IF rtbTrigger.Q OR bKeepTryingMove OR bTriggerCounter THEN
		bTriggerCounter := FALSE; 
		bKeepTryingMove := FALSE;
		nFormCounter := 0;
		bBottlePresent:= bCapPresent  := FALSE; 
		
			FOR j:=1 TO 3 DO
				FOR i:= 1 TO iExitArrayElements-1 DO // SORTOWANIE
					IF NOT eExitState[i].bFormPresent THEN 
						eExitState[i] := eExitState[i+1];
						eExitState[i+1] := eClearPackageState;
					END_IF
				END_FOR
			END_FOR	
		
			FOR i := 1 TO iEntranceArrayElements DO
				IF  NOT eExitState[i].bFormPresent THEN  		// Jeżeli w rejestrze wyjściowym jest wolne miejsce to wpisz rejestr wejściowy
					eExitState[i] := eEntranceState[1];	// Wpisz do rejestru dane np z [1] Buffor do [1,2,3,4,5,6] Package
					eEntranceState[1]:=eClearPackageState;	// Czyszczenie pierwszego rejestru wejściowego
					k:=i;											// Przepisywanie zmiennej pomocniczej
					FOR i := 1 TO iEntranceArrayElements DO   				
						IF i = iEntranceArrayElements THEN
							eEntranceState[i]:=eClearPackageState;		  // Zerowanie ostatniego bo zostało przesuniete wszystko o 1
						ELSE													  // Przepisanie 2 do 1, 3 do 2, 4 do 3, 5 do 4, 6 do 5, zeruj 6
							eEntranceState[i] := eEntranceState[i+1]; // 2 do 1, 3 do 2,
							eEntranceState[i+1]:=eClearPackageState;		  // zeruj 2, 
						END_IF
					END_FOR
					bTriggerDone := TRUE;
					EXIT;
					bError := TRUE;
					iError := 1;
				ELSE
					nFormCounter := nFormCounter + 1;
					bError := TRUE;
					iError := 2;
				END_IF
			END_FOR
		
		IF nFormCounter = iExitArrayElements THEN
		bKeepTryingMove:=NOT bNoKeepTryingMove;
		END_IF
	END_IF


//CZYSZCZENIE REJESTRU WEJSCIOWEGO
IF rtbReset.Q THEN
	FOR r1 := 1 TO iEntranceArrayElements DO
		eEntranceState[r1] := eClearPackageState;
	END_FOR
	FOR r2 := 1 TO iExitArrayElements DO
		eExitState[r2] := eClearPackageState;
	END_FOR
	bKeepTryingMove :=FALSE;
	bTriggerDone := FALSE;
	bTriggerCounter := FALSE; 
	nFormCounter := 0;
	bBottlePresent := bCapPresent := FALSE; 
	bError := FALSE;
	iError := 0;
END_IF

END_FUNCTION_BLOCK

// ---- POUs/FB/FB_InputFilter_v2.TcPOU
(*
Nazwa:			FB_InputFilter_v2
Opis: 			Filtrowanie czujnikow
Wersja:			v1.1
Data:			2023-09-20
Autor:			DP
Urzadzenia:		
Konfiguracja:	
Info:
- blok filtrujacy wejście cyfrowe
*)

FUNCTION_BLOCK FB_InputFilter_v2
VAR_INPUT
	bIN:BOOL;				//Wejście cyfrowe
	tFilterTimeOn:TIME;		//Czas filtrowania
	tFilterTimeOff:TIME;	//Czas filtrowania
END_VAR
VAR_OUTPUT
	bOUT:BOOL;
END_VAR
VAR
	tonIN: TON;
	tonOFF: TON;
END_VAR


(* w2 *)
tonIN	(IN:=bIN, 		PT:=tFilterTimeOn);
tonOFF	(IN:=NOT bIN, 	PT:=tFilterTimeOff);
IF tonIN.Q THEN
	bOUT := 	TRUE;
ELSIF tonOFF.Q THEN
	bOUT := 	FALSE;
END_IF

END_FUNCTION_BLOCK

// ---- POUs/FB/FB_MoveRegisterSortAndMoveROPP.TcPOU
(*
Nazwa:			FB_MoveRegister
Opis:			Blok przesuniecia rejestru formatek
Wersja:			v0.3 		
Data:			2018-11-16
Autor:			DP
Urzadzenia:		 
Konfiguracja:	
Info:
- Są dwa rejestry, wejściowy i wyjsciowy (struktury)
- Jezeli rejestr ma np. 6 elementów to za kazdym razem po wykryciu trigera program będzie
	1 wejściowy przesuwał na 1 wolny (nie ma formatki) wyjściowy
	kasował 1 rejestr wejściowy
	przesuwal rejetr wejsciowy 2 na 1(przeniesiony i skasowany), 3 na 2, 4 na 3, 5 na 4, 6 na 5 i kasowal 6wejsciowy
	tym sposobem po 6 trigerach caly rejestr wejsciowy powinien być na wyjsciowym
	np po 3 trigerach na wyjsciowym powinny byc zajete 1 do 3 i na wejsciowym 1 do 3
Błędy:
1 - nie wyszło z pętli for
2 - formatka już jest w rejestrze
Uwagi:
- 
Zmiany:
2018-09-18 Dodano sprawdzanie nasadek
2018-06-14 DP Pierwsza wersja
*)

FUNCTION_BLOCK FB_MoveRegisterSortAndMoveROPP
VAR_INPUT
	bFirstCycle:BOOL;					//Pierwszy cykl, zeby na początku nie wykrywało zbocza opadającego
	bTrigger :BOOL;						// Przesuniecie tablicy o jeden
	tTriggerFilterTimeOn:TIME:=T#0MS;	// Czas filtrowania wejścia Trigger na załączenie
	tTriggerFilterTimeOff:TIME:=T#0MS;	// Czas filtrowania wejścia Trigger na wyłączenie
	bTriggerBottle :BOOL;				// Zapisywanie czy jest butelka czy nie (jezeli kontrola wlączona)
	bWithBottleControl: BOOL;			// Włączona opcja kontroli butelek
	bWithCapControl:BOOL;				// Wlaczona kontrola nasadek
	bWithFormControlTrigerCounter:BOOL;	// Jezeku na trigercontrol nie ma formatki do przesunięcia to stwórz nową
	bMoveOnlyIfFormPresent:BOOL;		// Przepisuj tylko jak jest formatka
	bRotateEntranceRegisterBefore:BOOL;	// Najpierw przesuń rejestr wejściowy a następnie z niego zabierz
	bNoKeepTryingMove:BOOL;				// Dalej przepisuj jezeli nie ma miejsca
	bTriggerCap: BOOL;					// Truger wykrycia nasadki
	bReset :BOOL;						// Czyszczenie tablic
	iEntranceArrayElements :UINT; 		// Wartość koncowa tablicy
	iExitArrayElements :UINT; 			// Wartość koncowa tablicy
	bInvertWriting :BOOL;				// Wpisywanie odwrotne zamist z 1entrance na 1exit to 1entrance na 6exit	
	eClearPackageState :S_PackageState; // Czysty rejestr
END_VAR
VAR_IN_OUT
	bTriggerCounter :BOOL;		// Triger ktory jest kasowany
	eEntranceState :ARRAY [1..17] OF S_PackageState;	
	eExitState :ARRAY [1..17] OF S_PackageState;
	bKeepTryingMove :BOOL;		// Probuj dalej zapisać formatki aż się któraś zwolni
END_VAR

VAR_OUTPUT	
	bError :BOOL; 				// Błąd
	iError: UINT;				// Nr Błędu
	bTriggerDone :BOOL; 		// Wykonano przesunięcie
	bTriggerFilteredOUT:BOOL;	//Wyjscie przefiltrowanego sygnalu wejsciowego
END_VAR

VAR
	i:UINT;						// Zmienna w tablicy
	k:UINT;						// Pomocnicza zmienna do zapisywnia czy jest butelka
	rtbTrigger :R_TRIG;			// Reaguje na zbocze
	rtbTriggerBottle :R_TRIG;	// Reaguje na zbocze
	rtbReset :R_TRIG;			// Reaguje na zbocze
	TimerResetErrors :TON;		// Reset Błedu
	nFormCounter :UINT;					//Licznik formatek
	r1,r2:UINT;
	bBottlePresent: BOOL;				//Zmienna pomocnicza ze wykryto butelkę
	bCapPresent: BOOL;					//Zmienna pomocnicza ze wykryto butelkę
	j: UINT;
	tonTriggerFilterTimeOn: TON;
	bTriggerFiltered: BOOL;
	tofTriggerFilterTimeOff: TOF;
END_VAR

//Filtrowanie sygnału wejściowego
tofTriggerFilterTimeOff	(IN:=bTrigger, PT:=tTriggerFilterTimeOff);
tonTriggerFilterTimeOn	(IN:=tofTriggerFilterTimeOff.Q, PT:=tTriggerFilterTimeOn);
bTriggerFiltered 		:= tonTriggerFilterTimeOn.Q;
bTriggerFilteredOUT		:= bTriggerFiltered ;

//TRIGI I TIMERY
IF bWithBottleControl THEN
	rtbTrigger 	(CLK := NOT bTriggerFiltered, Q=>);
	rtbTriggerBottle 	(CLK := NOT bTriggerBottle, Q=>);
ELSIF bWithCapControl THEN
	rtbTrigger 	(CLK := NOT bTriggerFiltered, Q=>);
ELSE
	rtbTrigger 	(CLK := bTriggerFiltered, Q=>);
	rtbTriggerBottle 	(CLK := bTriggerBottle, Q=>);
END_IF

rtbReset 	(CLK := bReset, Q=>);
TimerResetErrors (IN:= bError, PT:=T#1000MS, Q=>);

//RESETOWANIE BLEDU
IF TimerResetErrors.Q THEN
	bError := FALSE;
END_IF

//KASOWANIE ZMIENNYCH
bTriggerDone := FALSE;

//JEZELI WLACZONO KONTROLE BUTELEK TO NADPISUJ REJESTR CZY JEST BUTELKA
IF bWithBottleControl AND bTrigger AND bTriggerBottle AND NOT bKeepTryingMove THEN //Jezeli od wykrycia formatki liczy TIMER i wykryło butelke to wpisz do rejestru że jest butelka
	eEntranceState[1].bBottlePresent := TRUE;
	eEntranceState[1].bFormPresent := TRUE;
	bBottlePresent := TRUE; // Wpisuje że jest butelka jezeli wystąpi sygnał podczas trwania czujnika formatki
ELSIF bWithBottleControl AND rtbTrigger.Q AND NOT bBottlePresent AND  NOT bKeepTryingMove AND bFirstCycle THEN
	eEntranceState[1].bBottlePresent := FALSE;
	eEntranceState[1].bFormPresent := TRUE; // jeżeli zanik czujnik formatki i nie było formatki to wpisz ze nie było butelki
END_IF

IF bWithCapControl AND bTriggerCap AND NOT bKeepTryingMove THEN //Jezeli od wykrycia formatki liczy TIMER i wykryło butelke to wpisz do rejestru że jest butelka
	eEntranceState[1].bCapPutted := TRUE;
	eEntranceState[1].bCapOK := TRUE; eEntranceState[1].bBottlePresent:= TRUE;//Zmiana nowa
	eEntranceState[1].bFormPresent := TRUE;
	bCapPresent := TRUE; // Wpisuje że jest butelka jezeli wystąpi sygnał podczas trwania czujnika formatki	
ELSIF bWithCapControl AND rtbTrigger.Q AND NOT bCapPresent AND  NOT bKeepTryingMove AND bFirstCycle THEN
	eEntranceState[1].bCapPutted := TRUE;
	eEntranceState[1].bCapOK:= FALSE;
	eEntranceState[1].bFormPresent := TRUE; // jeżeli zanik czujnik formatki i nie było formatki to wpisz ze nie było butelki
END_IF
//JEZELI WLACZONO SPRAWDZANIE FORMATEK Z TRIGERCOUNTER TO
IF bWithFormControlTrigerCounter  AND bTriggerCounter AND NOT bKeepTryingMove AND bFirstCycle THEN
	eEntranceState[1].bFormPresent := TRUE;
END_IF


//PRZESUNIECIE
IF (*iEntranceArrayElements <= iExitArrayElements AND*) bFirstCycle  THEN
		IF rtbTrigger.Q OR bKeepTryingMove OR bTriggerCounter THEN
		bTriggerCounter := FALSE; 
		bKeepTryingMove := FALSE;
		nFormCounter 	:= 0;
		bBottlePresent := bCapPresent  := FALSE; 
		FOR i:= 1 TO iExitArrayElements-1 DO // SORTOWANIE
			IF NOT eExitState[i].bFormPresent THEN 
				eExitState[i] := eExitState[i+1];
				eExitState[i+1] := eClearPackageState;
			END_IF
		END_FOR

		FOR i := 1 TO iExitArrayElements DO
			IF  NOT eExitState[i].bFormPresent THEN  		// Jeżeli w rejestrze wyjściowym jest wolne miejsce to wpisz rejestr wejściowy
				eExitState[i] := eEntranceState[1];			// Wpisz do rejestru dane np z [1] Buffor do [1,2,3,4,5,6] Package
				eEntranceState[1]:=eClearPackageState;		// Czyszczenie pierwszego rejestru wejściowego
				k:=i;										// Przepisywanie zmiennej pomocniczej
				FOR i := 1 TO iEntranceArrayElements DO   				
					IF i = iEntranceArrayElements THEN
						eEntranceState[i]:=eClearPackageState;			// Zerowanie ostatniego bo zostało przesuniete wszystko o 1
					ELSE												// Przepisanie 2 do 1, 3 do 2, 4 do 3, 5 do 4, 6 do 5, zeruj 6
						eEntranceState[i] := eEntranceState[i+1]; 		// 2 do 1, 3 do 2,
						eEntranceState[i+1]:= eClearPackageState;		// zeruj 2, 
					END_IF
				END_FOR
				bTriggerDone := TRUE;
				EXIT;
				bError := TRUE;
				iError := 5;
			ELSE
				nFormCounter := nFormCounter + 1;
				bError := TRUE;
				iError := 6;
			END_IF
		END_FOR

		IF nFormCounter = iExitArrayElements THEN
			bKeepTryingMove:=NOT bNoKeepTryingMove;
		END_IF
	END_IF
END_IF


//CZYSZCZENIE REJESTRU WEJSCIOWEGO
IF rtbReset.Q THEN
	FOR r1 := 1 TO iEntranceArrayElements DO
		eEntranceState[r1] := eClearPackageState;
	END_FOR
	FOR r2 := 1 TO iExitArrayElements DO
		eExitState[r2] := eClearPackageState;
	END_FOR
	bKeepTryingMove :=FALSE;
	bTriggerDone := FALSE;
	bTriggerCounter := FALSE; 
	nFormCounter := 0;
	bBottlePresent := bCapPresent := FALSE; 
	bError := FALSE;
	iError := 0;
END_IF

END_FUNCTION_BLOCK

// ---- POUs/FB/FB_MoveRegisterROPPCapControl.TcPOU
(*
Nazwa:			FB_MoveRegister
Opis:			Blok przesuniecia rejestru formatek
Wersja:			v0.3 		
Data:			2018-11-16
Autor:			DP
Urzadzenia:		 
Konfiguracja:	
Info:
- Są dwa rejestry, wejściowy i wyjsciowy (struktury)
- Jezeli rejestr ma np. 6 elementów to za kazdym razem po wykryciu trigera program będzie
	1 wejściowy przesuwał na 1 wolny (nie ma formatki) wyjściowy
	kasował 1 rejestr wejściowy
	przesuwal rejetr wejsciowy 2 na 1(przeniesiony i skasowany), 3 na 2, 4 na 3, 5 na 4, 6 na 5 i kasowal 6wejsciowy
	tym sposobem po 6 trigerach caly rejestr wejsciowy powinien być na wyjsciowym
	np po 3 trigerach na wyjsciowym powinny byc zajete 1 do 3 i na wejsciowym 1 do 3
Błędy:
1 - nie wyszło z pętli for
2 - formatka już jest w rejestrze
Uwagi:
- 
Zmiany:
2018-09-18 Dodano sprawdzanie nasadek
2018-06-14 DP Pierwsza wersja
*)

FUNCTION_BLOCK FB_MoveRegisterROPPCapControl
VAR_INPUT
	bFirstCycle:BOOL;					//Pierwszy cykl, zeby na początku nie wykrywało zbocza opadającego
	bTrigger :BOOL;						// Przesuniecie tablicy o jeden
	tTriggerFilterTimeOn:TIME:=T#0MS;	// Czas filtrowania wejścia Trigger na załączenie
	tTriggerFilterTimeOff:TIME:=T#0MS;	// Czas filtrowania wejścia Trigger na wyłączenie
	bTriggerBottle :BOOL;				// Zapisywanie czy jest butelka czy nie (jezeli kontrola wlączona)
	bWithBottleControl: BOOL;			// Włączona opcja kontroli butelek
	bWithCapControl:BOOL;				// Wlaczona kontrola nasadek
	bWithFormControlTrigerCounter:BOOL;	// Jezeku na trigercontrol nie ma formatki do przesunięcia to stwórz nową
	bNoKeepTryingMove:BOOL;				// Dalej przepisuj jezeli nie ma miejsca
	bTriggerCap: BOOL;					// Truger wykrycia nasadki
	bReset :BOOL;						// Czyszczenie tablic
	iEntranceArrayElements :UINT; 		// Wartość koncowa tablicy
	iExitArrayElements :UINT; 			// Wartość koncowa tablicy
	eClearPackageState :S_PackageState; // Czysty rejestr
END_VAR
VAR_IN_OUT
	eEntranceState :ARRAY [1..17] OF S_PackageState;	
	eExitState :ARRAY [1..17] OF S_PackageState;
	iBottleWithoutCap: INT;
	bKeepTryingMove :BOOL;		// Probuj dalej zapisać formatki aż się któraś zwolni
	bRFIDReaded :BOOL;
END_VAR

VAR_OUTPUT	
	bError :BOOL; 				// Błąd
	iError: UINT;				// Nr Błędu
	bTriggerDone :BOOL; 		// Wykonano przesunięcie

	bTriggerFilteredOUT:BOOL;	//Wyjscie przefiltrowanego sygnalu wejsciowego
END_VAR

VAR
	i:UINT;						// Zmienna w tablicy
	k:UINT;						// Pomocnicza zmienna do zapisywnia czy jest butelka
	rtbTrigger :R_TRIG;			// Reaguje na zbocze
	rtbTriggerBottle :R_TRIG;	// Reaguje na zbocze
	rtbReset :R_TRIG;			// Reaguje na zbocze
	TimerResetErrors :TON;		// Reset Błedu
	nFormCounter :UINT;					//Licznik formatek
	r1,r2:UINT;
	bBottlePresent: BOOL;				//Zmienna pomocnicza ze wykryto butelkę
	bCapPresent: BOOL;					//Zmienna pomocnicza ze wykryto butelkę
	j: UINT;
	tonTriggerFilterTimeOn: TON;
	bTriggerFiltered: BOOL;
	tofTriggerFilterTimeOff: TOF;
	fbTriggerFiltered: FB_InputFIlter;
	ftfbTriggerFiltered: F_TRIG;
	tpTrigger: TP;
END_VAR

//Filtrowanie sygnału wejściowego
fbTriggerFiltered		(bIN:= 	bTrigger AND bRFIDReaded,		tFilterTimeOn:=tTriggerFilterTimeOn,	tFilterTimeOff:=tTriggerFilterTimeOff);

//TRIGI I TIMERY
ftfbTriggerFiltered		(CLK:=	fbTriggerFiltered.bOUT, 	Q=>);

rtbReset 				(CLK := bReset, Q=>);
TimerResetErrors 		(IN:= bError, PT:=T#1000MS, Q=>);

//RESETOWANIE BLEDU
IF TimerResetErrors.Q THEN
	bError := FALSE;
END_IF

//KASOWANIE ZMIENNYCH
bTriggerDone := FALSE;

//JEZELI WLACZONO KONTROLE NASADEk TO NADPISUJ REJESTR CZY JEST BUTELKA 
IF bWithCapControl AND bTriggerCap AND NOT bKeepTryingMove THEN //Jezeli od wykrycia formatki liczy TIMER i wykryło butelke to wpisz do rejestru że jest butelka
	eEntranceState[1].bROPPPuttedChecked := TRUE;
	eEntranceState[1].bROPPPutted := TRUE; eEntranceState[1].bBottlePresent:= TRUE;//Zmiana nowa
	bCapPresent := TRUE; // Wpisuje że jest butelka jezeli wystąpi sygnał podczas trwania czujnika formatki	
ELSIF bWithCapControl AND ftfbTriggerFiltered.Q AND NOT bCapPresent AND  NOT bKeepTryingMove AND bFirstCycle THEN
	eEntranceState[1].bROPPPuttedChecked := TRUE;
	eEntranceState[1].bROPPPutted:= FALSE;
END_IF


//PRZESUNIECIE
IF iEntranceArrayElements < iExitArrayElements AND bFirstCycle THEN
	IF ftfbTriggerFiltered.Q OR bKeepTryingMove THEN
		bRFIDReaded		:= FALSE;
		bKeepTryingMove := FALSE;
		nFormCounter 	:= 0;
	
		IF bCapPresent THEN		
			eEntranceState[1].bROPPPuttedChecked := TRUE;
			eEntranceState[1].bROPPPutted := TRUE; eEntranceState[1].bBottlePresent:= TRUE;
			eEntranceState[1].bFormPresent := TRUE;
		END_IF

		bBottlePresent := bCapPresent  := FALSE; 
		
		FOR i:= 1 TO iExitArrayElements-1 DO // SORTOWANIE PRZED
			IF NOT eExitState[i].bFormPresent THEN 
				eExitState[i] := eExitState[i+1];
				eExitState[i+1] := eClearPackageState;
			END_IF
		END_FOR
		
		FOR i := 1 TO iExitArrayElements DO
			IF  NOT eExitState[i].bFormPresent THEN  		// Jeżeli w rejestrze wyjściowym jest wolne miejsce to wpisz rejestr wejściowy
				eExitState[i] 		:= 	eEntranceState[1];	// Wpisz do rejestru dane np z [1] Buffor do [1,2,3,4,5,6] Package
				eEntranceState[1]	:=	eClearPackageState;	// Czyszczenie pierwszego rejestru wejściowego
				k:=i;										// Przepisywanie zmiennej pomocniczej
				bTriggerDone := TRUE;
				IF eExitState[i].bBottlePresent AND NOT eExitState[i].bROPPPutted THEN
					iBottleWithoutCap	:=	iBottleWithoutCap	+1;
				END_IF
				IF eExitState[i].bBottlePresent AND eExitState[i].bROPPPutted THEN
					iBottleWithoutCap	:=	0;	
				END_IF	
				IF NOT eExitState[i].bBottlePresent THEN
					iBottleWithoutCap	:=	0;	
				END_IF				
				EXIT;
				bError := TRUE;
				iError := 5;
			ELSE
				nFormCounter := nFormCounter + 1;
				bError := TRUE;
				iError := 6;
			END_IF
		END_FOR
		IF nFormCounter = iExitArrayElements THEN
			bKeepTryingMove:=NOT bNoKeepTryingMove;
		END_IF
	END_IF
END_IF

//CZYSZCZENIE REJESTRU WEJSCIOWEGO
IF rtbReset.Q THEN
	FOR r1 := 1 TO iEntranceArrayElements DO
		eEntranceState[r1] := eClearPackageState;
	END_FOR
	FOR r2 := 1 TO iExitArrayElements DO
		eExitState[r2] := eClearPackageState;
	END_FOR
	bKeepTryingMove :=FALSE;
	bTriggerDone := FALSE;
	nFormCounter := 0;
	bBottlePresent := bCapPresent := FALSE; 
	bError := FALSE;
	iError := 0;
END_IF

END_FUNCTION_BLOCK

// ---- POUs/FB/FB_AutoTrialRenew_ADS.TcPOU
FUNCTION_BLOCK FB_AutoTrialRenew_ADS
VAR_INPUT
    bExpired            : BOOL;          // sygnał końca licencji (Twój)
    sProductId          : STRING(80);    // ID licencji Beckhoff
    sAdsServerNetId     : STRING(40);    // AMS ID serwera licencji
    nAdsServerPort      : UINT := 10000; // port ADS serwera
END_VAR

VAR_OUTPUT
    bBusy               : BOOL;
    bDone               : BOOL;
    bError              : BOOL;
    nErrorId            : UDINT;

    sLicenseOut         : STRING(1024);  // nowa licencja trial
END_VAR

VAR
    fbAdsWrite          : AdsWrite;
    fbAdsRead           : AdsRead;

    eState              : INT := 0;
    sBuffer             : STRING(1024);
END_VAR

// ============================================================================
//  STATE MACHINE
// ============================================================================
CASE eState OF

// ------------------------------------------------------
// IDLE
// ------------------------------------------------------
0:
    bBusy := FALSE;
    bDone := FALSE;
    bError := FALSE;

    IF bExpired THEN
        bBusy := TRUE;
        eState := 10;
    END_IF

// ------------------------------------------------------
// SEND REQUEST (ADS WRITE) – send ProductId to ADS server
// ------------------------------------------------------
10:
	fbAdsWrite(
		NETID	:=sAdsServerNetId,
		PORT	:=nAdsServerPort,
		IDXGRP	:=16#80000001,
		IDXOFFS	:=0,
		LEN		:=SIZEOF(sProductId),
		SRCADDR	:=ADR(sProductId),
		WRITE	:=TRUE);
		

    IF fbAdsWrite.ERR THEN
        bError := TRUE;
        nErrorId := fbAdsWrite.ERRID;
        eState := 0;

    ELSIF NOT fbAdsWrite.BUSY (*AND NOT fbAdsWrite.WRITE*) THEN
        eState := 20;
    END_IF

// ------------------------------------------------------
// GET TRIAL LICENCE (ADS READ)
// ------------------------------------------------------
20:
	fbAdsRead(
		NETID	:=sAdsServerNetId,
		PORT	:=nAdsServerPort, 
		IDXGRP	:=16#80000002,
		IDXOFFS	:=0,
		LEN		:=SIZEOF(sBuffer),
        DESTADDR:=ADR(sBuffer),
        READ	:=TRUE);
		
    IF fbAdsRead.ERR THEN
        bError := TRUE;
        nErrorId := fbAdsRead.ERRID;
        eState := 0;

    ELSIF NOT fbAdsRead.BUSY (*AND NOT fbAdsRead.READ *)THEN
        sLicenseOut := sBuffer;
        bDone := TRUE;
        bBusy := FALSE;
        eState := 0;
    END_IF

END_CASE

END_FUNCTION_BLOCK

// ---- POUs/P00_SystemDiagnostics.TcPOU
//==================================================================================================
//							Beckhoff Automation Poland
//									2.11.2018
//					Program zbiorczy diagnostyki systemu
// 
//	v1.4 	|| TC v 3.1.4022.25 	|| Dodany state machine
//	v1.3 	|| TC v 3.1.4022.20 	|| Usuniete P_MDP, dodany podprogram EventLoggera P_SystemDiag_EventLog
//	v1.2 	|| TC v 3.1.4020.32 	|| Dodane P_EtherCAT_ChangeCounter
//	v1.1 	|| TC v 3.1.4020.14 	|| Dodane wyjscia bOk, bWarning, bError
//	v1.0 	|| TC v 3.1.4020.0 		|| Pierwsza wersja
//==================================================================================================
PROGRAM P00_SystemDiagnostics
VAR_INPUT
	bReset													: BOOL;
END_VAR                                     				
VAR_OUTPUT                                  				
	eDiagState												: E_DiagState;
	bOK														: BOOL;									// Brak bledow i ostrzezen
	bWarning												: BOOL;									// Ostrzezenie
	bError													: BOOL;									// Zbiorcza flaga bledow
	udiErrorID												: UDINT;								// Numer bledu
	sErrorDescription										: WSTRING;								// Opis blad
END_VAR                                     	
VAR                                         	
	tonCheckDiagnosisResettingTime							: TON;									// Timer do zabezpieczenia zeby program nie utknal w ressetingu
	iEtherCatDiagResetStep									: INT;
	fb_EtherCatReqMasterState								: FB_EcReqMasterState;
	sAmsNetID_EtherCATMaster								: T_AmsNetId := '192.168.40.180.3.1';	// EtherCAT Master AMS Net ID
	fbGetStateRobot 										: FB_EcGetSlaveState;
	rtstatequest 											: R_TRIG;
END_VAR

P_SystemInfo();																												// Wywolanie programow sprawdzajacych
P_Persistent();
P_EtherCAT_Diag();
P_EtherCAT_ChangeCounter();
P_Checks();
P_TaskInfo();
P_PlcTaskSystemInfo();							
P_GroupsWcStates();


bError													:= //	P_SystemInfo.bError 				OR 
															//P_Persistent.bError 				OR 
															{warning {'chwilowo wykOMENTAOWANE, ODKOMENTOWAĆ!'}//P_EtherCAT_Diag.bError 				OR
															P_EtherCAT_ChangeCounter.bError 	OR 
															P_Checks.bError 					OR 
															//P_TaskInfo.bError 					OR 
														(*	P_PlcTaskSystemInfo.bError 			OR *)
															P_GroupsWcStates.bError;
                                                		
bWarning												:= //	P_SystemInfo.bWarning 				OR 
															// P_Persistent.bWarning 				OR 
															P_EtherCAT_Diag.bWarning 			OR 
															P_EtherCAT_ChangeCounter.bWarning 	OR 
															P_Checks.bWarning 				;//	OR 
															// P_TaskInfo.bWarning 			(*	OR 
															//P_PlcTaskSystemInfo.bWarning*);
													
bOk															:= NOT (bError OR bWarning);

rtstatequest(CLK:=bError);

IF P_SystemInfo.bError OR P_SystemInfo.bWarning THEN																			// Przypisanie numerow bledow oraz opisow do zmiennych 
	udiErrorID												:= P_SystemInfo.udiErrorID; 										// Bledy od 1-4
	sErrorDescription										:= P_SystemInfo.sErrorDescription;	
	                                            			
ELSIF P_Persistent.bError THEN                  			
	udiErrorID												:= P_Persistent.udiErrorID;
	sErrorDescription										:= P_Persistent.sErrorDescription;
	                                            			
ELSIF P_EtherCAT_Diag.bError THEN               			
	udiErrorID												:= P_EtherCAT_Diag.udiErrorID;        
	sErrorDescription										:= P_EtherCAT_Diag.sErrorDescription;	
	
ELSIF P_EtherCAT_ChangeCounter.bError THEN
	udiErrorID												:= P_EtherCAT_ChangeCounter.udiErrorID;
	sErrorDescription										:= P_EtherCAT_ChangeCounter.sErrorDescription;	
	                                            			
ELSIF P_Checks.bError THEN                      			
	udiErrorID												:= P_Checks.udiErrorID;        
	sErrorDescription										:= P_Checks.sErrorDescription;	
                                                			
ELSIF P_TaskInfo.bError THEN                    			
	udiErrorID												:= P_TaskInfo.udiErrorID;       
	sErrorDescription										:= P_TaskInfo.sErrorDescription;
	                                            			
ELSIF P_PlcTaskSystemInfo.bError THEN           			
	udiErrorID												:=  P_PlcTaskSystemInfo.udiErrorID;       
	sErrorDescription										:=  P_PlcTaskSystemInfo.sErrorDescription;
	                                            	
ELSIF P_GroupsWcStates.bError THEN              	
	udiErrorID												:= P_GroupsWcStates.udiErrorID; 									// Bledy od 10-11
	sErrorDescription										:= P_GroupsWcStates.sErrorDescription;
	
ELSIF NOT bError THEN
	udiErrorID												:= 0;
	sErrorDescription										:= "";	
END_IF


// State machine
CASE eDiagState OF

	///////////////
	E_DiagState.eOK:
	
		IF bError OR P_SystemInfo.bWarning THEN
			eDiagState										:= E_DiagState.eError;
		END_IF
		
	///////////////////		
	E_DiagState.eError:

		IF bReset THEN
			eDiagState										:= E_DiagState.eResetting;
			bReset := FALSE;
		END_IF
		//wyjście ze stanu błędu jak wszystko ok
		IF bOk THEN 
			eDiagState										:= E_DiagState.eOK;
		END_IF
			
	//////////////////////
	E_DiagState.eResetting:

		(*Program P_EtherCAT_Diag automatycznie przyjmuje stan OK lub Error w zaleznosci od stanu modulow*)
		P_EtherCAT_ChangeCounter.bReset						:= NOT P_EtherCAT_ChangeCounter.bOK;
		P_Checks.bReset										:= NOT P_Checks.bOK;
		P_Persistent.bReset									:= NOT P_Persistent.bOK;
		P_TaskInfo.bReset									:= NOT P_TaskInfo.bOK;
		P_SystemInfo.bReset									:= P_SystemInfo.bError OR P_SystemInfo.bWarning;
		P_PlcTaskSystemInfo.bReset							:= NOT P_PlcTaskSystemInfo.bOK;
		P_GroupsWcStates.bReset								:= NOT P_GroupsWcStates.bOK;																	
		//reset ethercat w przypadku błędu sieci
		IF P_EtherCAT_Diag.bError AND iEtherCatDiagResetStep=0 THEN
			iEtherCatDiagResetStep							:= 10;
		END_IF
		
		IF NOT bError THEN 
			P_EtherCAT_ChangeCounter.bReset					:= FALSE;
		    P_Checks.bReset									:= FALSE;
		    P_Persistent.bReset								:= FALSE;
		    P_TaskInfo.bReset								:= FALSE;
		    P_SystemInfo.bReset								:= FALSE;
		    P_PlcTaskSystemInfo.bReset						:= FALSE;
		    P_GroupsWcStates.bReset							:= FALSE;
			iEtherCatDiagResetStep							:= 0;
			eDiagState										:= E_DiagState.eOK;
		END_IF
		
		IF bError AND tonCheckDiagnosisResettingTime.Q THEN														// Jesli pomimo resetu dalej jest blad przejsie do statu eError
			
			P_EtherCAT_ChangeCounter.bReset					:= FALSE;											// Kasowanie zmiennych od resetu programow sprawdzajacych
		    P_Checks.bReset									:= FALSE;
		    P_Persistent.bReset								:= FALSE;
		    P_TaskInfo.bReset								:= FALSE;
		    P_SystemInfo.bReset								:= FALSE;
			P_PlcTaskSystemInfo.bReset						:= FALSE;
			P_GroupsWcStates.bReset							:= FALSE;
			iEtherCatDiagResetStep							:= 0;
			eDiagState:= E_DiagState.eError;
		END_IF
	
END_CASE
	
// Log to events - You can switch it off in Initialization phase
P_SystemDiag_EventLog();


CASE iEtherCatDiagResetStep OF
	0:	//Oczekiwanie na reset
		fb_EtherCatReqMasterState.sNetId			:= sAmsNetID_EtherCATMaster;
		fb_EtherCatReqMasterState.bExecute			:= FALSE;
		fb_EtherCatReqMasterState.tTimeout			:= T#5S;
		fb_EtherCatReqMasterState.state				:= EC_DEVICE_STATE_INIT;
		//EC_DEVICE_STATE_INIT			0x01		Request Init state from master
		//EC_DEVICE_STATE_PREOP			0x02		Request Pre-operational state from master
		//EC_DEVICE_STATE_SAFEOP		0x04		Request Safe-operational state from master
		//EC_DEVICE_STATE_OP			0x08		Request Operational state from master
		
	10:	//wynuś INIT
		fb_EtherCatReqMasterState.bExecute			:= TRUE;
		fb_EtherCatReqMasterState.state				:= EC_DEVICE_STATE_INIT;
		IF fb_EtherCatReqMasterState.bBusy THEN
			fb_EtherCatReqMasterState.bExecute		:= FALSE;
			iEtherCatDiagResetStep					:= 20;
		END_IF
	20:
		IF NOT fb_EtherCatReqMasterState.bBusy THEN
			fb_EtherCatReqMasterState.state			:= EC_DEVICE_STATE_OP;
			iEtherCatDiagResetStep					:= 30;
		END_IF
	30: //wymuś OP
		fb_EtherCatReqMasterState.bExecute			:= TRUE;
		IF fb_EtherCatReqMasterState.bBusy THEN
			fb_EtherCatReqMasterState.bExecute		:= FALSE;
			iEtherCatDiagResetStep					:= 40;
		END_IF
	40:
		IF NOT fb_EtherCatReqMasterState.bBusy THEN
			iEtherCatDiagResetStep					:= 0;
			eDiagState								:= E_DiagState.eOK;
		END_IF
		
END_CASE

fb_EtherCatReqMasterState();

tonCheckDiagnosisResettingTime.IN							:= eDiagState = E_DiagState.eResetting AND iEtherCatDiagResetStep = 0; 					// Uzywane do kasowania resetu na poszczegolnych podprogramach
tonCheckDiagnosisResettingTime.PT							:= T#400MS;												 		// patrz case Resetting(zrobione po to aby kiedy utrzyma sie blad
tonCheckDiagnosisResettingTime();                       																	// przejsc do casu error




//Vasyl diagnostyka robota 03.10

fbGetStateRobot(
    sNetId     := sAmsNetID_EtherCATMaster,       // '' = lokalnie
    nSlaveAddr := 1049,         // adres EtherCAT slave
    bExecute   := rtstatequest.q
);

END_PROGRAM

// ---- POUs/FB/Diagnostics/POUsDiagnosticComponents/P_SystemInfo.TcPOU
//==================================================================================================
//							Beckhoff Automation Poland
//									P_SystemInfo
//									31.10.2018
//					Program odczytujący informacje o TC Runtime
// 
//	v1.2 	|| TC v 3.1.4022.25 	|| - bOK dodane BSOD i sprawdzenie licencji
//	v1.1 	|| TC v 3.1.4020.14 	|| - Dodane wyjscia bOk, bWarning, bError
//	v1.0 	|| TC v 3.1.4020.0 		|| - Pierwsza wersja
//==================================================================================================
PROGRAM P_SystemInfo
VAR_INPUT
	bConfirm					: BOOL;					// Potwierdzenie bledu/ostrzezenia persistentow - blad/ostrzezenie nie znika, my usuwamy flage error lub warning
	bReset						: BOOL;
END_VAR
VAR_OUTPUT
	bOK							: BOOL;					// Zmienne wczytane prawidlowo
	bWarning					: BOOL;					// Zmienne wczytane z pliku zapasowego
	bError						: BOOL;					// Nie wczytano zmiennych
	sErrorDescription			: WSTRING;
	udiErrorID					: UDINT;
END_VAR
VAR
	sStartTime					: STRING;				// Przekonwertowany czas
	rtReset						: R_TRIG;
	bFirstCycle: BOOL;
END_VAR

rtReset(CLK:= bReset);

IF rtReset.Q AND bWarning THEN
	bConfirm					:= TRUE;
END_IF

//_AppInfo.ObjId; 			(* Object ID of the PLC project instance *)
//_AppInfo.TaskCnt;			(* The number of tasks in the actual runtime system *)
//_AppInfo.OnlineChangeCnt;	(* The number of online changes made since the last complete download. *)
//_AppInfo.Flags;				(* Reserved for future use *)
//_AppInfo.AdsPort; 			(* ADS port of PLC application *)
bOK							:= (_AppInfo.BootDataLoaded OR bConfirm) AND NOT _AppInfo.LicensesPending AND NOT _AppInfo.BSODOccured;	(* PERSISTENT variables: LOADED (without error) *)
bWarning					:= _AppInfo.OldBootData AND NOT bConfirm;	(* PERSISTENT variables: INVALID (the back-up copy was loaded, since no valid data was present) *)
bError						:= NOT bOK AND NOT bWarning AND bFirstCycle;
//_AppInfo.KeepOutputsOnBP;	(* The flag can be set to avoid that the outputs are zero-filled if a breakpoint is reached. The task keeps running. Only the execution of PLC code is interrupted. *)
//_AppInfo.TComSrvPtr;		(* Pointer to TcCOM Object Server *)
//_AppInfo.AppName;			(* TwinCAT generated name containing the port number. *)
//_AppInfo.ProjectName;		(* The name of the PLC project. *)
sStartTime					:= DELETE(DT_TO_STRING(_AppInfo.AppTimestamp),3,1);(* Date and time of application start *)
(*_AppInfo.BSODOccured;
_AppInfo.LicensesPending;
_AppInfo.ShutdownInProgress;*)

IF bOK THEN
	sErrorDescription			:= "";
	udiErrorID					:= 0;
END_IF


IF bError OR bWarning THEN
	IF _AppInfo.LicensesPending THEN
		sErrorDescription		:= "Błąd sterownika | Oczekiwanie na licencję sterownika";
		udiErrorID				:= 92;
	ELSIF _AppInfo.OldBootData AND bWarning THEN
		sErrorDescription		:= "Błąd sterownika | Załadowano nieaktualne dane sterownika";
		udiErrorID				:= 93;
	ELSIF _AppInfo.BSODOccured THEN
		sErrorDescription		:= "Błąd sterownika | Wystąpił BlueScreenOfDeath";
		udiErrorID				:= 94;
	ELSE
		sErrorDescription		:= "Błąd sterownika | Błąd wczytania danych sterownika";
		udiErrorID				:= 95;
	END_IF
END_IF

bFirstCycle:= TRUE;

END_PROGRAM

// ---- POUs/FB/Diagnostics/POUsDiagnosticComponents/P_Persistent.TcPOU
//==================================================================================================
//							Beckhoff Automation Poland
//									25.04.2018
//		Program obslugujacy pamiec nieulotna 
//	v1.4    || TC v 3.1.4026.19		|| - Obsługa UPS
// 	v1.3	|| TC v 3.1.4022.16		|| - Przeniesienie logowania do EvenLogger'a do programu P_SystemDiag_EventLog
// 	v1.2	|| TC v 3.1.4022.0		|| - Dodanie akcji UPS
//	v1.1 	|| TC v 3.1.4020.14 	|| - Dodane wyjscia bOk, bWarning, bError
//	v1.0 	|| TC v 3.1.4020.0 		|| - Pierwsza wersja
//==================================================================================================
PROGRAM P_Persistent
VAR_INPUT
	sAmsNetID_EtherCATMaster	: T_AmsNetId	:= '192.168.40.160.3.1';			// EtherCAT Master AMS Net ID
	bWritePersistent			: BOOL;
	bReset						: BOOL;
END_VAR
VAR_OUTPUT
	bOK							: BOOL 						:= TRUE;				// Brak bledow i ostrzezen
	bWarning					: BOOL;												// Ostrzezenie
	bError						: BOOL;												// Zbiorcza flaga bledow
	udiErrorID					: UDINT;
	sErrorDescription			: WSTRING;
	bWrited						: BOOL;
	bPowerFailDetect			: BOOL;
END_VAR
VAR																			
	iStep						: INT;
	fbWritePersistentData		: FB_WritePersistentData;
	
	//fbUPS						: FB_S_UPS;
	//fbUPS_CB3011				: FB_S_UPS_CB3011;
	fbUPS_CX51x0				: FB_S_UPS_CX51x0;
	//fbUPS_CX9020_U900			: FB_S_UPS_CX9020_U900;
	//fbUPS_BAPI					: FB_S_UPS_BAPI;
	fbUPS_CU8130				:FB_GetUPSStatus;
	
	eUpsMode					: E_S_UPS_Mode;
	eUpsState					: E_S_UPS_State;
	
	
	iNumberOfWrites				: INT;
	rtWritePersistent			: R_TRIG;
END_VAR


ACT_UPS();
ACT_WritePersistent();

fbUPS_CU8130.stStatus.ePowerStatus;
fbUPS_CU8130.stStatus.eBatteryStatus;
fbUPS_CU8130.stStatus.nPowerFailCnt;
fbUPS_CU8130.stStatus.eCommStatus;
IF fbUPS_CU8130.stStatus.ePowerStatus=2 AND NOT bWrited THEN
	bWritePersistent:=TRUE;
ELSE
	bWritePersistent:=FALSE;
END_IF

ACTION A_fbS_UPS:
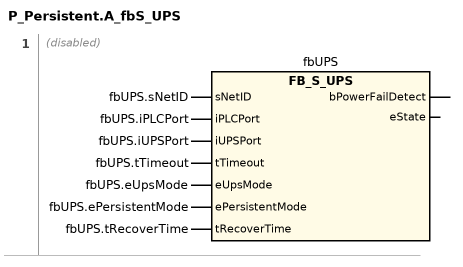
// NETWORK 1 (disabled)
// fbUPS(
//     sNetID := fbUPS.sNetID,
//     iPLCPort := fbUPS.iPLCPort,
//     iUPSPort := fbUPS.iUPSPort,
//     tTimeout := fbUPS.tTimeout,
//     eUpsMode := fbUPS.eUpsMode,
//     ePersistentMode := fbUPS.ePersistentMode,
//     tRecoverTime := fbUPS.tRecoverTime); // FB_S_UPS
END_ACTION

ACTION A_fbS_UPS_BAPI:
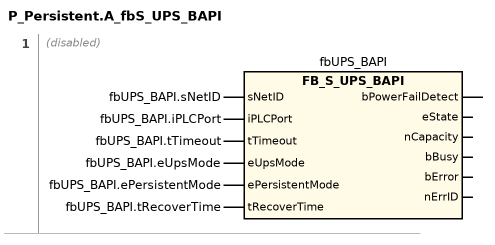
// NETWORK 1 (disabled)
// fbUPS_BAPI(
//     sNetID := fbUPS_BAPI.sNetID,
//     iPLCPort := fbUPS_BAPI.iPLCPort,
//     tTimeout := fbUPS_BAPI.tTimeout,
//     eUpsMode := fbUPS_BAPI.eUpsMode,
//     ePersistentMode := fbUPS_BAPI.ePersistentMode,
//     tRecoverTime := fbUPS_BAPI.tRecoverTime); // FB_S_UPS_BAPI
END_ACTION

ACTION A_fbS_UPS_CB3011:
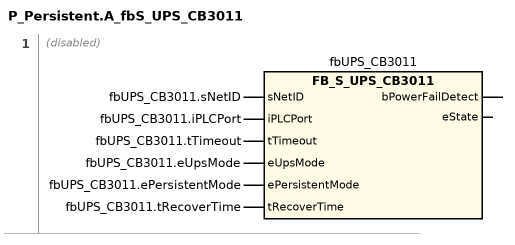
// NETWORK 1 (disabled)
// fbUPS_CB3011(
//     sNetID := fbUPS_CB3011.sNetID,
//     iPLCPort := fbUPS_CB3011.iPLCPort,
//     tTimeout := fbUPS_CB3011.tTimeout,
//     eUpsMode := fbUPS_CB3011.eUpsMode,
//     ePersistentMode := fbUPS_CB3011.ePersistentMode,
//     tRecoverTime := fbUPS_CB3011.tRecoverTime); // FB_S_UPS_CB3011
END_ACTION

ACTION A_fbS_UPS_CX51x0:
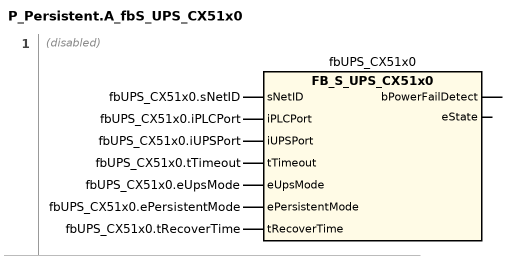
// NETWORK 1 (disabled)
// fbUPS_CX51x0(
//     sNetID := fbUPS_CX51x0.sNetID,
//     iPLCPort := fbUPS_CX51x0.iPLCPort,
//     iUPSPort := fbUPS_CX51x0.iUPSPort,
//     tTimeout := fbUPS_CX51x0.tTimeout,
//     eUpsMode := fbUPS_CX51x0.eUpsMode,
//     ePersistentMode := fbUPS_CX51x0.ePersistentMode,
//     tRecoverTime := fbUPS_CX51x0.tRecoverTime); // FB_S_UPS_CX51x0
END_ACTION

ACTION A_fbS_UPS_CX9020_U900:
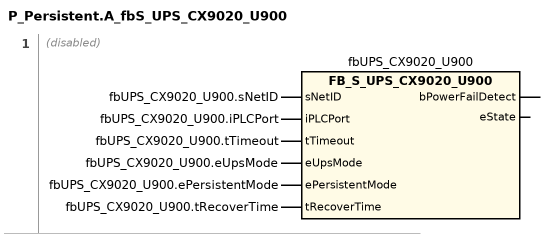
// NETWORK 1 (disabled)
// fbUPS_CX9020_U900(
//     sNetID := fbUPS_CX9020_U900.sNetID,
//     iPLCPort := fbUPS_CX9020_U900.iPLCPort,
//     tTimeout := fbUPS_CX9020_U900.tTimeout,
//     eUpsMode := fbUPS_CX9020_U900.eUpsMode,
//     ePersistentMode := fbUPS_CX9020_U900.ePersistentMode,
//     tRecoverTime := fbUPS_CX9020_U900.tRecoverTime); // FB_S_UPS_CX9020_U900
END_ACTION

ACTION ACT_UPS:
//fbUPS_CX9020_U900
//(
//	sNetID							:= sAmsNetID_EtherCATMaster, 
//	iPLCPort						:= 851, 
//	tTimeout						:= DEFAULT_ADS_TIMEOUT, 
//	eUpsMode						:= E_S_UPS_Mode.eSUPS_WrPersistData_Shutdown,
//	ePersistentMode					:= E_PersistentMode.SPDM_2PASS, 
//	tRecoverTime					:= T#10S, 
//	bPowerFailDetect				=> bPowerFailDetect, 
//	eState							=> eUpsState
//);


//fbUPS_CX51x0
//(
//	sNetID							:= sAmsNetID_EtherCATMaster, 
//	iPLCPort						:= 851, 
//	iUPSPort						:= 16#588, 
//	tTimeout						:= DEFAULT_ADS_TIMEOUT, 
//	eUpsMode						:= E_S_UPS_Mode.eSUPS_WrPersistData_Shutdown, 
//	ePersistentMode					:= E_PersistentMode.SPDM_2PASS, 
//	tRecoverTime					:= T#10S, 
//	bPowerFailDetect				=> bPowerFailDetect, 
//	eState							=> eUpsState
//);
fbUPS_CU8130
(	sNetID							:='',
	nPort							:=0,
	bEnable							:=TRUE,
	bValid							=>,
	bError	=>,
	nErrId =>,
	stStatus =>,);
END_ACTION

ACTION ACT_WritePersistent:
rtWritePersistent(CLK:= bWritePersistent);


CASE iStep OF

0:
	IF rtWritePersistent.Q THEN
		fbWritePersistentData.PORT												:= _AppInfo.AdsPort;
		fbWritePersistentData.MODE												:= SPDM_2PASS;	
		fbWritePersistentData.START												:= TRUE;
		bWrited																	:= FALSE;
		iStep:= 10;
	END_IF

10:
	IF NOT fbWritePersistentData.BUSY THEN
		IF NOT fbWritePersistentData.ERR THEN
			fbWritePersistentData.START											:= FALSE;
			bWrited																:= TRUE;	
			iNumberOfWrites														:= iNumberOfWrites + 1;
			iStep:= 20;
		END_IF
	END_IF

	IF fbWritePersistentData.ERR THEN
 	
		bWrited																	:= FALSE;
		bError																	:= TRUE;	
		udiErrorID																:= fbWritePersistentData.ERRID;
		sErrorDescription														:= "Błąd zapisu zmiennych PERSISTENT";
		iStep:= 900;
	END_IF
	
20:
	IF NOT bWritePersistent THEN
		iStep:= 0;
	END_IF	
	
900:
	bOK																			:= FALSE;
	
	IF bReset THEN
		fbWritePersistentData.START												:= FALSE;
	END_IF
	IF NOT bReset THEN
		fbWritePersistentData.START												:= TRUE;
	END_IF
	
	
	IF NOT fbWritePersistentData.BUSY THEN
		IF NOT fbWritePersistentData.ERR THEN 
			bOK																	:= TRUE;
			bError																:= FALSE;
			udiErrorID															:= 0;
			sErrorDescription													:= "";
			iStep:= 0;	
		END_IF
	END_IF
	

END_CASE


fbWritePersistentData();
END_ACTION

END_PROGRAM

// ---- POUs/FB/Diagnostics/POUsDiagnosticComponents/P_EtherCAT_Diag.TcPOU
//==================================================================================================
//							Beckhoff Automation Poland
//									18.06.2018
//		Program wysyłający błędy magistrali EBus do EvenLogger'a
//
//	v1.4	|| TC v 3.1.4022.16		|| - Przeniesiono logowanie do EventLoggera wraz z zabepieczeniem przed zbyt szybkim logowaniem zdarzeń do programu P_SystemDiag_EventLog. 
//	v1.3	|| TC v 3.1.4020.28		|| - Dodano zabezpieczenie przed zbyt sczęstym logowaniem eventów i zmieniono system logowania błędów ramek. Od teraz każda ramka ma swój EventId. Wstępnie zarezerwowano 8 ramek.
//  v1.2	|| TC v 3.1.4020.28		|| - Usunięto zbędne wejścia (sFormat, pDataAdr i udiDataLen) na fbDevDiag które podoowały generowanie błędów przekroczeń indeksów
//									|| - Dodano logowanie do EventLoggera 
//	v1.1 	|| TC v 3.1.4020.14 	|| - Dodane wyjscia bOk, bWarning, bError
//	v1.0 	|| TC v 3.1.4020.0 		|| - Pierwsza wersja
//==================================================================================================
PROGRAM P_EtherCAT_Diag
VAR CONSTANT
	iNumOfFrames				: INT := 6;						// Liczba FrmWcState
END_VAR
VAR_OUTPUT
	bOK							: BOOL;								// Brak bledow i ostrzezen
	bWarning					: BOOL;								// Ostrzezenie - nie wystepuja w tym podprogramie - wystepuja dla zachowania spojnosci
	bError						: BOOL;								// Zbiorcza flaga bledow
	udiErrorID					: UDINT;	
	sErrorDescription			: WSTRING;
END_VAR
VAR
	uiDevState		AT %I*		: UINT;								// DevState mastera EtherCAT'a
																	(*	0x0001 = Link error
																		0x0002 = I/O locked after link error (I/O reset required)
																		0x0004 = Link error (redundancy adapter)
																		0x0008 = Missing one frame (redundancy mode)
																		0x0010 = Out of send resources (I/O reset required)
																		0x0020 = Watchdog triggered
																		0x0040 = Ethernet driver (miniport) not found
																		0x0080 = I/O reset active
																		0x0100 = At least one device in 'INIT' state
																		0x0200 = At least one device in 'PRE-OP' state
																		0x0400 = At least one device in 'SAFE-OP' state
																		0x0800 = At least one device indicates an error state
																		0x1000 = DC not in sync*)
	uiFrmWcState		AT %I*	: ARRAY[1..iNumOfFrames] OF UINT;	// FrmWcState
																	(*	0x0001 = wrong working counter of 1. EtherCAT command received
																		0x0002 = wrong working counter of 2. EtherCAT command received
																		0x0004 = wrong working counter of 3. EtherCAT command received
																		...
																		...
																		0x4000 = wrong working counter of 15. EtherCAT command received
																		0x8000 = complete frame missing*)
	iIterator					: INT;
	rtError						: R_TRIG;
END_VAR

bError 									:= uiDevState <> 0;							// Ustawienie flagi bledu zgodnie z uiDevState

FOR iIterator := 1 TO iNumOfFrames DO
	IF uiFrmWcState[iIterator] <> 0 THEN
		bError 							:= TRUE;									// Ustawienie flagi bledu gdy chociaz jeden frame jest z bledem
		EXIT;
	END_IF
END_FOR


rtError									(CLK:= bError);

IF rtError.Q THEN
	udiErrorID							:= 97;	
	sErrorDescription					:= "Błąd sterownika | Błąd diagnostyki sieci EtherCAT";
END_IF

IF NOT bError THEN
	udiErrorID							:= 0;	
	sErrorDescription					:= "";
END_IF

bOK 									:= NOT bError AND NOT bWarning;

END_PROGRAM

// ---- POUs/FB/Diagnostics/POUsDiagnosticComponents/P_EtherCAT_ChangeCounter.TcPOU
//==================================================================================================
//							Beckhoff Automation Poland
//									19.10.2018
// Program wyświetlający informację o licznikach State Changes i NOT Present - opis ponizej
// Wymagane jest podanie jedynie adresu AMS NET ID Mastera EtherCATa i liczby urzadzen Slave
// State Changes/Not Present
// State Changes - for example if the sync task needs longer then 100ms, state changes from OP to other, but Slave is present
// Not Present - If it switchs back from OP (power off, broken...)
//
//	v1.3 	|| TC v 3.1.4022.25		 	|| - Reset as an input, Presen --> Present 
//	v1.2 	|| TC v 3.1.4022.20		 	|| - Return instruction and some comments
//	v1.1 	|| TC v 3.1.4020.32		 	|| - Dodane wyjscia bOk, bWarning, bError, opisu, zmiana typow zmiennych
//	v1.0 	|| TC v 3.1.4020.32 		|| - Pierwsza wersja
//==================================================================================================
PROGRAM P_EtherCAT_ChangeCounter
VAR CONSTANT
	sAmsNetID_EtherCATMaster				: T_AmsNetId	:= '192.168.40.180.3.1';		// EtherCAT Master AMS Net ID
	wCountOfEtherCATSlaves					: WORD 			:= 67; 							// Count of EtherCAT Slaves
END_VAR
VAR_INPUT
	bReset									: BOOL;
END_VAR
VAR_OUTPUT
	bOK										: BOOL;											// Brak bledow i ostrzezen
	bWarning								: BOOL;											// Ostrzezenie - nie wystepuja w tym podprogramie - wystepuja dla zachowania spojnosci
	bError									: BOOL;											// Zbiorcza flaga bledow
	udiErrorID								: UDINT;
	sErrorDescription						: WSTRING;
END_VAR
VAR
	//======================= State Changes/ ========================
	arrAbnormalStateChangeCounter			: ARRAY [1..wCountOfEtherCATSlaves] OF DWORD; 	// State Changes/  - tablica zawieraca dane dla poszczegilnych Slave
	wAbnormalStateChangeCounterPosition		: WORD;											// Pozycja pierwszego Slavea który zmienił wartosc licznika
	bAbnormalStateChangeCounterChanged		: BOOL;											// Flaga wystapienia zmiany licznika
	//===============================================================
	//======================== /Not Present =========================
	arrPresentStateChangeCounter			: ARRAY [1..wCountOfEtherCATSlaves] OF DWORD; 	// /Not Present  - tablica zawieraca dane dla poszczegilnych Slave
	wPresentStateChangeCounterPosition		: WORD;											// Pozycja pierwszego Slavea który zmienił wartosc licznika
	bPresentStateChangeCounterChanged		: BOOL;											// Flaga wystapienia zmiany licznika
	//===============================================================
	//======================= Internal ==============================
	bFirstCycle								: BOOL := TRUE;
	tonRefresh								: TON;
	tRefreshTime							: TIME := T#200MS;								// Refresh timer
	
	//===============================================================
	//=================== Internal hidden ===========================
	{attribute 'hide'}
	fbADSREAD_AbnormalStateChangeCounter	: ADSREAD;
	{attribute 'hide'}
	fbADSREAD_PresentStateChangeCounter		: ADSREAD;
	//{attribute 'hide'}
	arrAbnormalStateChangeCounterOld		: ARRAY [1..wCountOfEtherCATSlaves] OF DWORD; 	// Stara tablica - do celow porownawczych
	//{attribute 'hide'}
	arrPresenStateChangeCounterOld			: ARRAY [1..wCountOfEtherCATSlaves] OF DWORD; 	// Stara tablica - do celow porownawczych
	{attribute 'hide'}
	i										: WORD;
	{attribute 'hide'}
	ft1										: F_TRIG;
	{attribute 'hide'}
	ft2										: F_TRIG;
	//===============================================================
	rtReset: R_TRIG;
	rtError: R_TRIG;
END_VAR


{region "Is it ready to read?"}
IF sAmsNetID_EtherCATMaster = '' OR wCountOfEtherCATSlaves = 0 THEN
	RETURN;
END_IF
{endregion}
{region "Call FBs"}
// Start reading
tonRefresh(IN:= NOT tonRefresh.Q, PT:= tRefreshTime);

// End of reading 
ft1(CLK:= fbADSREAD_PresentStateChangeCounter.BUSY);
ft2(CLK:= fbADSREAD_AbnormalStateChangeCounter.BUSY);

// Reading
fbADSREAD_PresentStateChangeCounter(
	NETID			:= sAmsNetID_EtherCATMaster,
	PORT			:= 16#FFFF,
	IDXGRP			:= 16#16,
	IDXOFFS			:= 0,
	LEN				:= SIZEOF(arrPresentStateChangeCounter),
	DESTADDR		:= ADR(arrPresentStateChangeCounter),
	READ			:= tonRefresh.Q);

fbADSREAD_AbnormalStateChangeCounter(
	NETID			:= sAmsNetID_EtherCATMaster,
	PORT			:= 16#FFFF,
	IDXGRP			:= 16#13,
	IDXOFFS			:= 0,
	LEN				:= SIZEOF(arrAbnormalStateChangeCounter),
	DESTADDR		:= ADR(arrAbnormalStateChangeCounter),
	READ			:= ft1.Q);
{endregion}
{region "Change detection"}
//================= Checks positon of change ====================
// Check if changed
IF ft1.Q THEN
	IF NOT  bFirstCycle THEN
		FOR i := 1 TO wCountOfEtherCATSlaves DO
			IF arrPresentStateChangeCounter[i] <> arrPresenStateChangeCounterOld[i] THEN
				wPresentStateChangeCounterPosition 		:= i;
				bPresentStateChangeCounterChanged 		:= TRUE;
				EXIT;
			END_IF
		END_FOR
	END_IF
	arrAbnormalStateChangeCounterOld 					:= arrAbnormalStateChangeCounter;
END_IF

IF ft2.Q THEN
	IF NOT  bFirstCycle THEN
		FOR i := 1 TO wCountOfEtherCATSlaves DO
			IF arrAbnormalStateChangeCounter[i] <> arrAbnormalStateChangeCounterOld[i] THEN
				wAbnormalStateChangeCounterPosition 	:= i;
				bAbnormalStateChangeCounterChanged 		:= TRUE;
				EXIT;
			END_IF
		END_FOR
	END_IF
	arrPresenStateChangeCounterOld 						:= arrPresentStateChangeCounter;
	bFirstCycle 										:= FALSE;
END_IF
//===============================================================
{endregion}
{region "Reset and states"}
//  Reset
	 
rtReset(CLK:= bReset);
rtError(CLK:= bError);	
	  
IF rtReset.Q THEN
	wPresentStateChangeCounterPosition 					:= 0;
	wAbnormalStateChangeCounterPosition 				:= 0;
	bPresentStateChangeCounterChanged 					:= FALSE;
	bAbnormalStateChangeCounterChanged 					:= FALSE;
END_IF

// Set outputs
bError 													:= bPresentStateChangeCounterChanged OR bAbnormalStateChangeCounterChanged;
bOK 													:= NOT bError AND NOT bWarning;
	 
IF bError THEN
	udiErrorID											:= 98;
	sErrorDescription									:= "Błąd sterownika | Błąd jednego z urządzeń sieci EtherCAT";
ELSE
	udiErrorID											:= 0;
	sErrorDescription									:= "";		
END_IF	
		   
					
{endregion}

ACTION ACT_SlaveNames:
IF wPresentStateChangeCounterPosition 		= 1 THEN
;
ELSIF wPresentStateChangeCounterPosition 	= 2 THEN
;
ELSIF wPresentStateChangeCounterPosition 	= 3 THEN
;	
ELSIF wPresentStateChangeCounterPosition 	= 4 THEN
;	
ELSIF wPresentStateChangeCounterPosition 	= 5 THEN
;	
END_IF
END_ACTION

END_PROGRAM

// ---- POUs/FB/Diagnostics/POUsDiagnosticComponents/Checks/P_Checks.TcPOU
//==================================================================================================
//							Beckhoff Automation Poland
//									19.10.2018
//	Program wykrywajacy bledy dzielnia przez 0 i przekraczania zakresow zmiennych, tablic...
// 
//	v1.4	|| TC v 3.1.4022.25		|| - Ustawiono setowanie bledow, dodano wejscie bReset 
//	v1.3	|| TC v 3.1.4022.16		|| - Przeniesiono logowanie do EventLoggera wraz z zabepieczeniem przed zbyt szybkim logowaniem zdarzeń do programu P_SystemDiag_EventLog. 
//	v1.2	|| TC v 3.1.4020.28		|| - Dodano logowanie do EventLoggera wraz z zabepieczeniem przed zbyt szybki logowaniem zdarzeń
//	v1.1 	|| TC v 3.1.4020.14 	|| - Dodane wyjscia bOk, bWarning, bError
//	v1.0 	|| TC v 3.1.4020.0 		|| - Pierwsza wersja
//==================================================================================================
PROGRAM P_Checks
VAR_INPUT
	bReset							: BOOL;
END_VAR
VAR_OUTPUT
	bOK								: BOOL;	// Brak bledow i ostrzezen
	bWarning						: BOOL;	// Ostrzezenie - nie wystepuja w tym podprogramie - wystepuja dla zachowania spojnosci
	bError							: BOOL;	// Zbiorcza flaga bledow
	udiErrorID						: UDINT;       
	sErrorDescription				: WSTRING;
END_VAR
VAR
	bCheckBounds					: BOOL;	// Flaga przekroczen zakresu indexow, np. tablic
	bCheckDivDInt					: BOOL;	// Flaga prob dzielenia Dint przez 0
	bCheckDivLInt					: BOOL; // Flaga prob dzielenia LInt przez 0
	bCheckDivLReal					: BOOL; // Flaga prob dzielenia LREAL przez 0
	bCheckDivReal					: BOOL; // Flaga prob dzielenia REAL przez 0
	bCheckRangeSigned				: BOOL;	// Flaga przekroczen liczby znakowej
	bCheckRangeUnsigned				: BOOL; // Flaga przekroczen liczby bezznakowej
	
	dCheckBoundsOld					: DINT;	// Licznik przekroczen zakresu indexow, np. tablic
	dCheckDivDIntOld				: DINT;	// Licznik prob dzielenia Dint przez 0
	dCheckDivLIntOld				: DINT; // Licznik prob dzielenia LInt przez 0
	dCheckDivLRealOld				: DINT; // Licznik prob dzielenia LREAL przez 0
	dCheckDivRealOld				: DINT; // Licznik prob dzielenia REAL przez 0
	dCheckRangeSignedOld			: DINT;	// Licznik przekroczen  liczby znakowej
	dCheckRangeUnsignedOld			: DINT; // Licznik przekroczen  liczby bezznakowej
	
	rtError							: R_TRIG;
END_VAR

IF bReset THEN
	bCheckBounds 					:= FALSE;
	bCheckDivDInt					:= FALSE;
	bCheckDivLInt					:= FALSE;
	bCheckDivLReal					:= FALSE;
	bCheckDivReal					:= FALSE;
	bCheckRangeSigned				:= FALSE;
	bCheckRangeUnsigned				:= FALSE;
ELSE
	bCheckBounds 					S= dCheckBoundsOld <> gvlChecks.dCheckBounds;
	bCheckDivDInt					S= dCheckDivDIntOld <> gvlChecks.dCheckDivDInt;
	bCheckDivLInt					S= dCheckDivLIntOld <> gvlChecks.dCheckDivLInt;
	bCheckDivLReal					S= dCheckDivLRealOld <> gvlChecks.dCheckDivLReal;
	bCheckDivReal					S= dCheckDivRealOld <> gvlChecks.dCheckDivReal;
	bCheckRangeSigned				S= dCheckRangeSignedOld <> gvlChecks.dCheckRangeSigned;
	bCheckRangeUnsigned				S= dCheckRangeUnsignedOld <> gvlChecks.dCheckRangeUnsigned;	
END_IF

dCheckBoundsOld 					:= gvlChecks.dCheckBounds;
dCheckDivDIntOld 					:= gvlChecks.dCheckDivDInt;
dCheckDivLIntOld 					:= gvlChecks.dCheckDivLInt;
dCheckDivLRealOld 					:= gvlChecks.dCheckDivLReal;
dCheckDivRealOld 					:= gvlChecks.dCheckDivReal;
dCheckRangeSignedOld 				:= gvlChecks.dCheckRangeSigned;
dCheckRangeUnsignedOld 				:= gvlChecks.dCheckRangeUnsigned;

bError 								:= bCheckBounds OR bCheckDivDInt OR bCheckDivLInt OR bCheckDivLReal OR bCheckDivReal OR bCheckRangeSigned OR bCheckRangeUnsigned;
bOK 								:= NOT bError AND NOT bWarning;


rtError								(CLK:= bError);
                                    
IF rtError.Q THEN                   
	udiErrorID						:= 99;                         
	sErrorDescription				:= "Błąd sterownika | Błąd programu sprawdzającego operacje sterownika";	
END_IF                              
                                    
IF NOT bError THEN                  
	udiErrorID						:= 0;	
	sErrorDescription				:= "";
END_IF

END_PROGRAM

// ---- POUs/FB/Diagnostics/POUsDiagnosticComponents/P_TaskInfo.TcPOU
//==================================================================================================
//						Beckhoff Automation Poland
//							21.05.2018
//				Program  odczytujący informacje o tasku pierwszym.
//
// 	v1.1 || TC v 3.1.4022.16 || - zgodnosc ze standardem
// 	v1.0 || TC v 3.1.4020.14 || - pierwsza wersja
//==================================================================================================
PROGRAM P_TaskInfo
VAR_INPUT
	bReset						: BOOL;
END_VAR
VAR_OUTPUT
	bOK							: BOOL;						// Brak bledow i ostrzezen
	bWarning					: BOOL;						// Ostrzezenie - nie wystepuja w tym podprogramie - wystepuja dla zachowania spojnosci
	bError						: BOOL;						// Zbiorcza flaga bledow
	udiErrorID					: UDINT;
	sErrorDescription			: WSTRING;
END_VAR
VAR
	fbTaskInfo					: FB_TaskInfo;
	rtError						: R_TRIG;
END_VAR

bError 							:= fbTaskInfo.bError; 		// Dla jednego tasku. W przypadku wiekszej ilosci taskow trzeba dopisac reszte.
bOk 							:= NOT bError;
fbTaskInfo.bReset				:= bReset;


fbTaskInfo();


rtError									(CLK:= bError);

IF rtError.Q THEN
	udiErrorID							:= 96;                                            
	sErrorDescription					:= "Błąd sterownika | Błąd programu sprawdzającego cykl sterownik";	
END_IF

IF NOT bError THEN
	udiErrorID							:= 0;	
	sErrorDescription					:= "";
END_IF

END_PROGRAM

// ---- POUs/FB/Diagnostics/FBsDiagnostic/FB_TaskInfo.TcPOU
//==================================================================================================
//							Beckhoff Automation Poland
//							FB_TaskInfo
//							15.11.2016
//
//				Blok funkcyjny odczytujący informacje o tasku
//				Zapamiętuje maksymalne czasy wykonania oraz licznik przekroczeń
//
// 	v1.1 	|| TC v 3.1.4020.14 	|| - dodanie wyjsc
// 	v1.0 	|| TC v 3.1.4020.14 	|| - pierwsza wersja
//==================================================================================================
FUNCTION_BLOCK FB_TaskInfo
VAR_INPUT
	bReset					: BOOL;
END_VAR
VAR_OUTPUT
	bError					: BOOL;
END_VAR
VAR
	fbGetCurTaskIdx			: GETCURTASKINDEX;
	rLastExecTime			: REAL;
	rCycleTime				: REAL;
	uiPriority				: UINT;
	sTaskName				: STRING(63);
	bCycleTimeExceeded		: BOOL;
	rCycleCount				: REAL;
	rTotalTime				: REAL;
	rAverageCycleTime		: REAL;
	bResetVisu				: BOOL;
	byIndex					: BYTE;
END_VAR
VAR PERSISTENT
	udiCountExceedCycle		: UDINT; 						
	rMaxExecTime			: REAL;						
END_VAR

fbGetCurTaskIdx(index=>byIndex);

(*Odczyt czasu cyklu i ostatniego czasu wykonania*)
rCycleTime 					:= UDINT_TO_REAL(_TaskInfo[byIndex].CycleTime)/10000.0;
rLastExecTime 				:= UDINT_TO_REAL(_TaskInfo[byIndex].LastExecTime)/10000.0;
(*Zapamiętanie maksymalnego czasu wykonania*)
IF rLastExecTime > rMaxExecTime THEN 
	rMaxExecTime 			:= rLastExecTime;
END_IF

uiPriority					:= _TaskInfo[byIndex].Priority;
sTaskName					:= _TaskInfo[byIndex].TaskName;
bCycleTimeExceeded			:= _TaskInfo[byIndex].CycleTimeExceeded;
bError 						:= bCycleTimeExceeded; // Blad gdy czas cyklu przekroczony

(*Licznik przekroczeń czasu cyklu*)
IF _TaskInfo[byIndex].CycleTimeExceeded  THEN 
	udiCountExceedCycle 	:= udiCountExceedCycle + 1; 
END_IF
rCycleCount 				:= rCycleCount + 1;
rTotalTime 					:= rLastExecTime + rTotalTime;
rAverageCycleTime 			:= rTotalTime / rCycleCount;

(*Reset wyliczanych wartości*)
IF bReset OR bResetVisu THEN
	udiCountExceedCycle 	:= 0;
	rMaxExecTime 			:= 0;
	rTotalTime 				:= 0;
	rCycleCount 			:= 0;
	rAverageCycleTime 		:= 0;
	bReset 					:= FALSE;
END_IF

END_FUNCTION_BLOCK

// ---- POUs/FB/Diagnostics/POUsDiagnosticComponents/P_PlcTaskSystemInfo.TcPOU
// Program sprawdzajacy liczbe przekroczen czasu cyklu Task'a
PROGRAM P_PlcTaskSystemInfo
VAR_INPUT
	bReset								: BOOL;
END_VAR
VAR
	fbGetCurTaskIdx  					: GETCURTASKINDEX;
	bCycleTimeExeeded					: BOOL;
	rCounterCycleTimeExeeded			: REAL;
	rtCounterCycleTimeExeeded			: R_TRIG;
	rtReset								: R_TRIG;
	rtError								: R_TRIG;
	tonDelayAfterPowerOn: TON;
	bPowerOnDelay: BOOL;
END_VAR
VAR_OUTPUT
	bError								: BOOL;
	bOK									: BOOL;
	bWarning							: BOOL;
	udiErrorID							: UDINT;
	sErrorDescription					: WSTRING;
END_VAR

fbGetCurTaskIdx();
bCycleTimeExeeded 						:= _TaskInfo[fbGetCurTaskIdx.index].CycleTimeExceeded;

(*Dodane opóżnienie zliczania błędu po uruchomieniu maszyny*)
tonDelayAfterPowerOn					(IN:=NOT bPowerOnDelay,	PT:=T#5S);
IF tonDelayAfterPowerOn.Q THEN
	bPowerOnDelay	:=	TRUE;
END_IF

rtCounterCycleTimeExeeded				(CLK:= bCycleTimeExeeded AND bPowerOnDelay);
rtReset									(CLK:= bReset);

IF rtCounterCycleTimeExeeded.Q THEN
	rCounterCycleTimeExeeded			:= rCounterCycleTimeExeeded + 1;
END_IF	

IF rtReset.Q THEN
	rCounterCycleTimeExeeded 			:= 0;
END_IF

IF rCounterCycleTimeExeeded = 0 THEN
	P_PlcTaskSystemInfo.bError			:= FALSE;
	P_PlcTaskSystemInfo.bOK				:= TRUE;
END_IF

IF rCounterCycleTimeExeeded > 0 THEN
	P_PlcTaskSystemInfo.bError			:= TRUE;
	P_PlcTaskSystemInfo.bOK				:= FALSE;
END_IF


rtError									(CLK:= bError);

IF rtError.Q THEN
	udiErrorID							:= 91;                         
	sErrorDescription					:= "Błąd sterownika | Przekroczenie czasu cyklu";	
END_IF

IF NOT bError THEN
	udiErrorID							:= 0;	
	sErrorDescription					:= "";
END_IF

END_PROGRAM

// ---- POUs/FB/Diagnostics/POUsDiagnosticComponents/P_GroupsWcStates.TcPOU
PROGRAM P_GroupsWcStates
VAR_INPUT
	bReset															: BOOL;
	arrWcStateSyncUnitGroup	 				AT %I* 					: ARRAY [1..iNumberOfSyncUnitGroups] OF BOOL; (*Link to SyncUnit WcStates*)
END_VAR

VAR_OUTPUT
	bOK																: BOOL;
	bError															: BOOL;
	udiErrorID														: UDINT;
	sErrorDescription												: WSTRING;
END_VAR                                                     		
                                                            		
VAR                                                         	
	rtReset															: R_TRIG;
	bFirstCycle														: BOOL;
END_VAR                                                     	
                                                            	
VAR CONSTANT                                                	
	iNumberOfSyncUnitGroups											: INT:= 9;					// Deklaracja liczby grup SyncUnit
END_VAR

IF iNumberOfSyncUnitGroups = 0 OR NOT bFirstCycle THEN
	bFirstCycle															:= TRUE;
	RETURN;
END_IF

rtReset(CLK:= bReset);

FOR i:= 1 TO iNumberOfSyncUnitGroups DO
	IF arrWcStateSyncUnitGroup[i] THEN
		bError														:= TRUE;
		EXIT;                                               		
	END_IF                                                  		
END_FOR                                                     		
                                                            		
bOK																	:= NOT bError;	
                                                            		
                                                            		
IF arrWcStateSyncUnitGroup[1] THEN                          		
	udiErrorID														:= 84;
	sErrorDescription												:= "Błąd sterownika | Błąd komunikacji modułów komunikacyjnych";
END_IF   

IF arrWcStateSyncUnitGroup[2] THEN                          		
	udiErrorID														:= 85;
	sErrorDescription												:= "Błąd sterownika | Błąd komunikacji modułów I/O";
END_IF                                                 			
                                                        			
IF arrWcStateSyncUnitGroup[3] THEN                      			
	udiErrorID														:= 86;
	sErrorDescription												:= "Błąd sterownika | Błąd komunikacji grupy falowników";
END_IF 
                                                 		
IF arrWcStateSyncUnitGroup[4] THEN                      			
	udiErrorID														:= 87;
	sErrorDescription												:= "Błąd sterownika | Błąd komunikacji grupy modułów safety";
END_IF  
                                                      		
IF arrWcStateSyncUnitGroup[5] THEN                      			
	udiErrorID														:= 88;
	sErrorDescription												:= "Błąd sterownika | Błąd komunikacji grupy modułów pneumatycznych";
END_IF   

IF arrWcStateSyncUnitGroup[6] THEN                      			
	udiErrorID														:= 89;
	sErrorDescription												:= "Błąd sterownika | Błąd komunikacji grupy safety NC";
END_IF 

IF arrWcStateSyncUnitGroup[7] THEN                      			
	udiErrorID														:= 90;
	sErrorDescription												:= "Błąd sterownika | Błąd komunikacji grupy analogowych";
END_IF   
                                                  		
IF rtReset.Q THEN                                       		
	bError															:= FALSE;
	udiErrorID														:= 0;
	sErrorDescription												:= "";
END_IF

END_PROGRAM

// ---- POUs/FB/Diagnostics/POUsDiagnosticComponents/P_SystemDiag_EventLog.TcPOU
//==================================================================================================
//							Beckhoff Automation Poland
//									7.12.2018
//	Program logowanie do EventLoggera wraz z zabepieczeniem przed zbyt szybkim logowaniem zdarzen
//	Dziala tylko w polaczeniu z podprogramami i z blokami FB_AdvancedLogEvent, FB_AntiBlinkAlarmFilter
// 
//	v1.2	|| TC v 3.1.4022.25		|| Usuniecie wejscia bEnable
//	v1.1	|| TC v 3.1.4022.25		|| Dodane ACT_EtherCAT_ChangeCounter i Wejscie bEnable
//	v1.0	|| TC v 3.1.4022.20		|| Pierwsza wersja
//==================================================================================================
PROGRAM P_SystemDiag_EventLog
VAR
//======================== Checks ===============================
	fbBounds						: FB_AdvancedLogEvent;	// Logowanie wystapienia przekroczenia zakresu indexow
	fbDivDint						: FB_AdvancedLogEvent;	// Logowanie wystapienia proby dzielenia DINT przez 0
	fbDivLInt						: FB_AdvancedLogEvent;	// Logowanie wystapienia proby dzielenia LINT przez 0
	fbDivLReal						: FB_AdvancedLogEvent;	// Logowanie wsytapienia proby dzielenia LREAL przez 0
	fbDivReal						: FB_AdvancedLogEvent;	// Logowanie wystapienia proby dzielenia REAL przez 0
	fbRangeSigned					: FB_AdvancedLogEvent;	// Logowanie wystapienia przekroczenia liczby znakowej
	fbRangeUnsigned					: FB_AdvancedLogEvent;	// Logowanie wystapienia przekroczenia liczby bezznakowej
	
	fbBoundsBlockMessage			: FB_AdvancedLogEvent;	// Logowanie wystapienia przekroczenia zakresu indexow
	fbDivDintBlockMessage			: FB_AdvancedLogEvent;	// Logowanie wystapienia proby dzielenia DINT przez 0
	fbDivLIntBlockMessage			: FB_AdvancedLogEvent;	// Logowanie wystapienia proby dzielenia LINT przez 0
	fbDivLRealBlockMessage			: FB_AdvancedLogEvent;	// Logowanie wsytapienia proby dzielenia LREAL przez 0
	fbDivRealBlockMessage			: FB_AdvancedLogEvent;	// Logowanie wystapienia proby dzielenia REAL przez 0
	fbRangeSignedBlockMessage		: FB_AdvancedLogEvent;	// Logowanie wystapienia przekroczenia liczby znakowej
	fbRangeUnsignedBlockMessage		: FB_AdvancedLogEvent;	// Logowanie wystapienia przekroczenia liczby bezznakowej

//===============================================================
//======================= Persistent ============================
	ftPersistentSave				: F_TRIG;
	fbPersistentEventLoad			: FB_AdvancedLogEvent;
	fbPersistentEventSave			: FB_AdvancedLogEvent;
//===============================================================
//======================== EtherCAT =============================
	bEBusDiagLogPermission			: BOOL	:= TRUE;
	bEBusInitialized				: BOOL;
	iEBusIterator					: INT;
	(*DevDiag SourceID 901*)
	fbEBusDiag						: ARRAY[0..12] OF FB_AdvancedLogEvent;
	fbEtherCATStateChanged			: FB_AdvancedLogEvent;		// ID: 101
	fbEtherCATNotPresent			: FB_AdvancedLogEvent;		// ID: 102
	(*FrmWcState SourceID 902*)
	fbFrmWcDiag						: ARRAY[1..P_EtherCAT_Diag.iNumOfFrames] OF FB_AdvancedLogEvent;
	stFrmDiag						: ARRAY[1..P_EtherCAT_Diag.iNumOfFrames] OF ST_FrmWcDiag;
	fbString						: FB_FormatString;	(*Blok funkcyjny konwertujący FrmWcState na format binarny*)
	tArg							: T_Arg;
	//Filtrowanie zbyt częstego logowania
	fbEBusDiagFilter				: ARRAY[0..12] OF FB_AntiBlinkAlarmFilter;
	fbEBusDiagBlockMessage			: FB_AdvancedLogEvent;
	bFrmDiagLogPermission			: ARRAY[1..P_EtherCAT_Diag.iNumOfFrames] OF BOOL;
	fbFrmDiagFilter					: ARRAY[1..P_EtherCAT_Diag.iNumOfFrames] OF FB_AntiBlinkAlarmFilter;
	fbFrmDiagBlockMessage			: ARRAY[1..P_EtherCAT_Diag.iNumOfFrames] OF FB_AdvancedLogEvent;
//===============================================================
//========================== KBus ===============================
	fbKBusDiag						: ARRAY[0..15] OF FB_AdvancedLogEvent;
	nKbusIterator					: INT;
	bKBusDiagLogPermission			: BOOL := TRUE;
	fbKBusDiagFilter				: ARRAY[0..15] OF FB_AntiBlinkAlarmFilter;
	fbKBusDiagBlockMessage			: FB_AdvancedLogEvent;
//===============================================================
END_VAR

ACT_Checks();
ACT_PersistentLogs();
ACT_EtherCAT_Diag();
ACT_EtherCAT_ChangeCounter();

ACTION ACT_Checks:
fbBounds(
	bSetEvent		:= P_Checks.bCheckBounds,
	eEventClass 	:= TCEVENTCLASS_ALARM,
	bQuit			:= FALSE, 
	udiSourceID		:= 905, 
	udiEventID		:= 1);

fbDivDint(
	bSetEvent		:= P_Checks.bCheckDivDint,
	eEventClass 	:= TCEVENTCLASS_ALARM,
	bQuit			:= FALSE, 
	udiSourceID		:= 905, 
	udiEventID		:= 2);
	
fbDivLInt(
	bSetEvent		:= P_Checks.bCheckDivLInt,
	eEventClass 	:= TCEVENTCLASS_ALARM,
	bQuit			:= FALSE, 
	udiSourceID		:= 905, 
	udiEventID		:= 3);
	
fbDivLReal(
	bSetEvent		:= P_Checks.bCheckDivLReal,
	eEventClass 	:= TCEVENTCLASS_ALARM,
	bQuit			:= FALSE, 
	udiSourceID		:= 905, 
	udiEventID		:= 4);
	
fbDivReal(
	bSetEvent		:= P_Checks.bCheckDivReal,
	eEventClass 	:= TCEVENTCLASS_ALARM,
	bQuit			:= FALSE, 
	udiSourceID		:= 905, 
	udiEventID		:= 5);
	
fbRangeSigned(
	bSetEvent		:= P_Checks.bCheckRangeSigned,
	eEventClass 	:= TCEVENTCLASS_ALARM,
	bQuit			:= FALSE, 
	udiSourceID		:= 905, 
	udiEventID		:= 6);
	
fbRangeUnsigned(
	bSetEvent		:= P_Checks.bCheckRangeUnsigned,
	eEventClass 	:= TCEVENTCLASS_ALARM,
	bQuit			:= FALSE, 
	udiSourceID		:= 905, 
	udiEventID		:= 7);
END_ACTION

ACTION ACT_EtherCAT_ChangeCounter:
fbEtherCATStateChanged(	bSetEvent		:= P_EtherCAT_ChangeCounter.bAbnormalStateChangeCounterChanged, 
						bQuit			:= FALSE, 
						udiSourceID		:= 901, 
						udiEventID		:= 101, 
						sFormat			:= '%d', 
						eEventClass		:= TCEVENTCLASS_ALARM, 
						pDataAddress	:= ADR(P_EtherCAT_ChangeCounter.wAbnormalStateChangeCounterPosition), 
						udiDataLenght	:= SIZEOF(P_EtherCAT_ChangeCounter.wAbnormalStateChangeCounterPosition));

fbEtherCATNotPresent(	bSetEvent		:= P_EtherCAT_ChangeCounter.bPresentStateChangeCounterChanged, 
						bQuit			:= FALSE, 
						udiSourceID		:= 901, 
						udiEventID		:= 102, 
						sFormat			:= '%d', 
						eEventClass		:= TCEVENTCLASS_ALARM, 
						pDataAddress	:= ADR(P_EtherCAT_ChangeCounter.wPresentStateChangeCounterPosition), 
						udiDataLenght	:= SIZEOF(P_EtherCAT_ChangeCounter.wPresentStateChangeCounterPosition));
END_ACTION

ACTION ACT_EtherCAT_Diag:
// Wstępne zezwolenie na logowanie alarmów
IF NOT bEBusInitialized THEN
	FOR iEBusIterator := 1 TO P_EtherCAT_Diag.iNumOfFrames DO
		bFrmDiagLogPermission[iEBusIterator]	:= TRUE;
	END_FOR
	bEBusInitialized					:= TRUE;
END_IF

// DevState
FOR iEBusIterator := 0 TO 12 DO
	fbEBusDiag[iEBusIterator](
						bSetEvent		:= GETBIT32(P_EtherCAT_Diag.uiDevState,INT_TO_SINT(iEBusIterator)) AND bEBusDiagLogPermission,
						eEventClass 	:= TCEVENTCLASS_ALARM,
						bQuit			:= FALSE,
						udiSourceID		:= 901,
						udiEventID		:= INT_TO_UDINT(iEBusIterator + 1));
END_FOR

// FrmWcState
FOR iEBusIterator := 1 TO P_EtherCAT_Diag.iNumOfFrames DO
	stFrmDiag[iEBusIterator].iNum		:= iEBusIterator;
	IF P_EtherCAT_Diag.uiFrmWcState[iEBusIterator] <> 0 THEN
		tArg.cbLen						:= SIZEOF(P_EtherCAT_Diag.uiFrmWcState[iEBusIterator]);
		tArg.eType						:= ARGTYPE_UINT;
		tArg.pData						:= ADR(P_EtherCAT_Diag.uiFrmWcState[iEBusIterator]);
		fbString(sFormat := '%b', arg1 := tArg);
		stFrmDiag[iEBusIterator].sBin 	:= fbString.sOut;
	END_IF
	fbFrmWcDiag[iEBusIterator](
						bSetEvent		:= NOT(P_EtherCAT_Diag.uiFrmWcState[iEBusIterator] = 0) AND bFrmDiagLogPermission[iEBusIterator],
						eEventClass 	:= TCEVENTCLASS_ALARM,
						bQuit			:= FALSE, 
						udiSourceID		:= 902,
						udiEventID		:= INT_TO_UDINT(iEBusIterator),
						sFormat			:= '%d%s',
						pDataAddress	:= ADR(stFrmDiag[iEBusIterator]),
						udiDataLenght	:= SIZEOF(stFrmDiag[iEBusIterator]) );
END_FOR
END_ACTION

ACTION ACT_PersistentLogs:
IF _TaskInfo[1].FirstCycle THEN
	fbPersistentEventLoad.bSetEvent 			:= TRUE;
	IF _AppInfo.BootDataLoaded AND _AppInfo.OldBootData = FALSE THEN 	// wczytano poprawnie zmienne nieulotne
		fbPersistentEventLoad.udiEventID		:= 1;
		fbPersistentEventLoad.eEventClass		:= TCEVENTCLASS_MESSAGE;
	ELSIF _AppInfo.BootDataLoaded AND _AppInfo.OldBootData THEN 		// wczytano zmienne z kopii
		fbPersistentEventLoad.udiEventID		:= 2;
		fbPersistentEventLoad.eEventClass		:= TCEVENTCLASS_WARNING;
	ELSE //blad wczytania zmiennych
		fbPersistentEventLoad.udiEventID		:= 3;
		fbPersistentEventLoad.eEventClass		:= TCEVENTCLASS_ALARM;
	END_IF
ELSE
	//gdy nie wczytało zmiennych nieulotnych to wyswietlaj ostrzezenie w eventach aktywnych
	IF NOT (_AppInfo.BootDataLoaded = FALSE AND _AppInfo.OldBootData = FALSE) THEN
		fbPersistentEventLoad.bSetEvent			:= FALSE;
	END_IF
END_IF

fbPersistentEventLoad(udiSourceID := 900);

ftPersistentSave (CLK := P_Persistent.fbWritePersistentData.BUSY);
IF ftPersistentSave.Q THEN
	fbPersistentEventSave.bSetEvent 			:= TRUE;
	IF P_Persistent.fbWritePersistentData.ERR THEN
		fbPersistentEventSave.sFormat 			:= '%d';
		fbPersistentEventSave.udiEventID		:= 11;
		fbPersistentEventSave.eEventClass		:= TCEVENTCLASS_ALARM;
		fbPersistentEventSave.pDataAddress		:= ADR(P_Persistent.fbWritePersistentData.ERRID);
		fbPersistentEventSave.udiDataLenght		:= SIZEOF(P_Persistent.fbWritePersistentData.ERRID);
	ELSE
		fbPersistentEventSave.sFormat			:= '';
		fbPersistentEventSave.udiEventID		:= 10;
		fbPersistentEventSave.eEventClass		:= TCEVENTCLASS_MESSAGE;
	END_IF
ELSE
	fbPersistentEventSave.bSetEvent				:= FALSE;
END_IF

fbPersistentEventSave(udiSourceID:= 900);
END_ACTION

END_PROGRAM

// ---- POUs/FB/Diagnostics/FBsDiagnostic/FB_AdvancedLogEvent.TcPOU
//==================================================================================================
//							Beckhoff Automation Poland
//								FB_AdvancedLogEvent
//									16.11.2016
//				OPIS
//  v1.2 	|| TC v 3.1.4020.28		|| - uporzadkowanie zmiennych
//  v1.1 	|| TC v 3.1.4020.0 		|| - dodanie zmiennych wejsciowych bQuitRequired, bFBCleanup, udiEventState, bQuitAck, podpiecie zmiennych Error i ErrorID
// 	v1.0 	|| TC v 3.1.4020.0 		|| - pierwsza wersja
//==================================================================================================
FUNCTION_BLOCK FB_AdvancedLogEvent
VAR_INPUT
	(*Parametry do przekazania na blok ADSLOGEVENT*)
	bSetEvent						: BOOL;
	bQuit							: BOOL;
	udiSourceID						: UDINT; 				// nr bazy
	udiEventID						: UDINT; 				// nr zdarzenia
	sFormat							: STRING;				// jak mamy parametry to wstawiamy np: %s%d jeżeli nie mamy to zostawiamy puste pole
	eEventClass						: E_TcEventClass;		// klasa błędów
	pDataAddress					: POINTER TO BYTE;		// adress zmiennych parametrów, gdy korzystamy z sFormat
	udiDataLenght					: UDINT;				// dluglosc zmiennych parametrów, gdy korzystamy sFormat
	bQuitRequired					: BOOL := FALSE;
	bFbCleanup						: BOOL := FALSE;
END_VAR
VAR_OUTPUT
	bError							: BOOL;
	udiErrorID						: UDINT;
	udiEventState					: UDINT;
	bQuitAck						: BOOL;
END_VAR
VAR
	fbLogEvent						: ADSLOGEVENT;  		// Blok wysyłający event
	Event							: TcEvent;				// Konfiguracja eventu
END_VAR

Event.bQuitRequired			:= bQuitRequired;
Event.DataFormatStrAddress	:= ADR(sFormat);
Event.StreamType			:= TCEVENTSTREAM_SIMPLE;
Event.SourceId				:= udiSourceID;
Event.Id					:= udiEventID;
Event.Class					:= eEventClass;
Event.Flags					:= TCEVENTFLAG_LOG OR TCEVENTFLAG_SRCID;
Event.ProgId				:= 'TcEventFormatter.TcXmlFormatter';

fbLogEvent(
	NETID:= , 
	PORT:= 110, 
	Event:=bSetEvent , 
	EventQuit:= bQuit, 
	EventConfigData:= Event, 
	EventDataAddress:=pDataAddress , 
	EventDataLength:=udiDataLenght , 
	FbCleanup:= bFbCleanup, 
	TMOUT:= , 
	EventState=> udiEventState, 
	Err=> bError, 
	ErrId=> udiErrorID, 
	Quit=> bQuitAck);

END_FUNCTION_BLOCK

// ---- POUs/FB/Diagnostics/FBsDiagnostic/FB_AntiBlinkAlarmFilter.TcPOU
//==================================================================================================
//							Beckhoff Automation Poland
//								FB_AntiBlinkAlarmFilter
//									20.12.2016
//				Blok służący do wyłączania logowania zdarzeń które pojawiają się zbyt często
// 	v1.0 || TC v 3.1.4020.28 || - pierwsza wersja
//==================================================================================================
FUNCTION_BLOCK FB_AntiBlinkAlarmFilter
VAR_INPUT
	bEvent			: BOOL;		// Status zdarzenia
	tTime			: TIME;		// Zadane okno czasowe
	uiLimit			: UINT;		// Maksymalna liczba zdarzeń jaka może się pojawić w oknie czasowym
END_VAR
VAR_IN_OUT
	bPermission		: BOOL;		// Flaga zezwolenia na logowanie zdarzeń
END_VAR
VAR
	tStartTime		: TIME;		// Zmienna przechowująca czas rozpoczęcia zliczania
	uiActCount		: UINT;		// Aktualna wartość licznika
	rtEdge			: R_TRIG;	// Zbocze narastające
END_VAR

rtEdge(CLK:=bEvent);
IF rtEdge.Q THEN							// Blok podejmuje akcję w przypadku wystapienia zdarzenia
	IF uiActCount = 0 THEN	
		tStartTime		:= TIME();			// W przypadku gdy licznik wynosi zero, zapisywany jest czas rozpoczęcia zliczania
	END_IF
	uiActCount			:= uiActCount + 1;	// Inkrementacja licznika liczby zdarzeń
	IF uiActcount >= uiLimit THEN			// W przypadku gdy liczba zdarzeń osiągnie zadany limit, sprawdzany jest czas w jakim one wystapiły. Jeśli czas jest większy niż dopuszczalny, resetowana jest flaga zezwolenia
		IF TIME() - tStartTime < tTime THEN
			bPermission	:= FALSE;		
		END_IF
		uiActCount 		:= 0;
	END_IF
	IF NOT bPermission THEN
		uiActCount		:= 0;
	END_IF
END_IF;

END_FUNCTION_BLOCK

// ---- POUs/P00_Communication.TcPOU
PROGRAM P00_Communication
VAR

	fbCapSorterAdsRead		: FB_AdsCommunicationRead;
	fbBottleSorterAdsRead	: FB_AdsCommunicationRead;


	stCommunicationWriteCapSorterIN						: ST_Communication;
	stAdsCommunicationWriteBottleSorterIN				: ST_Communication; 

	
	//READ
	fbAdsCommunicationReadBottleSorter						: FB_AdsCommunicationRead;
	
	stAdsCommunicationReadCapSorterOUT						: ST_Communication;	//Odczytane zmienne z CapSorter
	stAdsCommunicationReadBottleSorterOUT					: ST_Communication;	//Odczytane zmienne z BottleSorter
	
	bAdsReadErrorCapSorter									: BOOL;
	bAdsReadErrorBottleSorter								: BOOL;
	
	bAdsReadBusyCapSorter									: BOOL;
	bAdsReadBusyBottleSorter								: BOOL;
	
	udiAdsReadErrorIDCapSorter								: UDINT;
	udiAdsReadErrorIDBottleSorter							: UDINT;

	iTestStartCounter										: INT;
	iCountTestNew											: INT;
	bCapSorterEmergencyStop									: BOOL;
	bBottleSorterEmergencyStop								: BOOL;
	bCapSorterRobotInPlaceProcess							: BOOL;
	bCapSorterRobotInPickProcess							: BOOL;
	bCapSorterPlaceDone										: BOOL;
	bCapSorterNotWaitingToCommand							: BOOL;						
	
	tonConveyor1CanMoveDelay								: TON;
	tonConveyor2CanMoveDelay								: TON;
	
	tpStartCycle											: TP;
		
	fbCyclicReadout: 										TON;
	fbEPRead:												 FB_ReadAdsSymByName;
	fbUPRead:												 FB_ReadAdsSymByName;
	

END_VAR

bBottleSorterDisable	:=GVL_IO.IbBottleSorterDisable;	//Wyłączane od kluczyka safety
bCapSorterDisable		:=GVL_IO.IbCapSorterDisable;	//Wyłączane od kluczyka safety

stBottleSorterRead.iWatchdog;
stCapSorterRead.iWatchdog;

ACT_BottleSorterAdsRead();
ACT_BottleSorterVariablesRead();
ACT_BottleSorterVariablesWrite();
ACT_CapSorterAdsRead();
ACT_CapSorterVariablesRead();
ACT_CapSorterVariablesWrite();
//ACT_EPAdsRead();
//ACT_UPAdsRead();

//tpStartCycle.IN	:= P00_PackML.rtStart.Q  OR P00_PackML.bCapSorterBottleSorterAutoStart;
tpStartCycle.IN		:= VIS.bAllowStart  OR P00_PackML.bCapSorterBottleSorterAutoStart;

tpStartCycle.PT		:= T#3S;
tpStartCycle();

ACTION ACT_BottleSorterAdsRead:
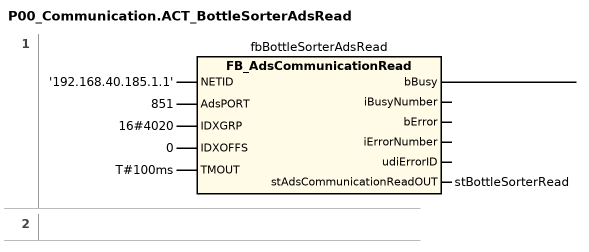
// NETWORK 1
fbBottleSorterAdsRead(
    NETID := '192.168.40.185.1.1',
    AdsPORT := 851,
    IDXGRP := 16#4020,
    IDXOFFS := 0,
    TMOUT := T#100ms,
    stAdsCommunicationReadOUT => stBottleSorterRead); // FB_AdsCommunicationRead

// NETWORK 2
END_ACTION

ACTION ACT_BottleSorterVariablesRead:
//PackMLState                                       		
stBottleSorterRead.ePackMLMode;
stBottleSorterRead.ePackMLAutoState; 
stBottleSorterRead.sPackMLCommand;
                      		
//stControlSignals        
stBottleSorterRead.bEnable;  bBottleSorterDisable;     // Potrzebujemy żeby odczytać czy stacja jest włączona w recepturach 
stBottleSorterRead.bCycleStart;
stBottleSorterRead.bCycleStop;
stBottleSorterRead.bCycleReset;
stBottleSorterRead.bManualMode;
stBottleSorterRead.bHoming;    // Wrote Homing przepisany w Sorterze na Read a w PackML robie bazowanie od Read
stBottleSorterRead.bHomingDone;	
stBottleSorterRead.bConfectionEnding;
stBottleSorterRead.tCycleTime;
stBottleSorterRead.iWatchdog;

//stError	
IF stBottleSorterRead.bEnable AND NOT bBottleSorterDisable THEN
	stBottleSorterRead.eError.bError;
ELSE
	stBottleSorterRead.eError.bError := FALSE;
END_IF

stBottleSorterRead.eError.bError;
stBottleSorterRead.eError.bReset;
stBottleSorterRead.eError.sErrorString;
stBottleSorterRead.eError.sStationName;
stBottleSorterRead.eError.nErrorCode;

//stRecipe
stBottleSorterRead.sRecipeName;
stBottleSorterRead.sRecipeIndex;
                             	                                 	
//stMachinePermissions                      	
bBottleSorterDoor1Open	:=	stBottleSorterRead.eMachinePermissions.bPermission00;	
bBottleSorterDoor2Open	:=	stBottleSorterRead.eMachinePermissions.bPermission01;
stBottleSorterRead.eMachinePermissions.bPermission02;	
stBottleSorterRead.eMachinePermissions.bPermission03;	
stBottleSorterRead.eMachinePermissions.bPermission04;	
stBottleSorterRead.eMachinePermissions.bPermission05;	
QbSafetyResetBottleSorterIn	:=	stBottleSorterRead.eMachinePermissions.bPermission06 AND NOT bBottleSorterDisable;;	//SafetyReset
bBottleSorterSystemDiagError := stBottleSorterRead.eMachinePermissions.bPermission07;	
//stBottleSorterRead.eMachinePermissions.bPermission10-17

//stReservedSignals
stBottleSorterRead.eReservedSignals.bReserved00;
stBottleSorterRead.eReservedSignals.bReserved01;
stBottleSorterRead.eReservedSignals.bReserved02; 
stBottleSorterRead.eReservedSignals.bReserved03; 
stBottleSorterRead.eReservedSignals.bReserved04;
stBottleSorterRead.eReservedSignals.bReserved05;
;stBottleSorterRead.eReservedSignals.bReserved06;
;stBottleSorterRead.eReservedSignals.bReserved07;
//stBottleSorterRead.eReservedSignals.bReserved10-17
stBottleSorterRead.eReservedSignals.iReserved20;//Warningi
stBottleSorterRead.eReservedSignals.iReserved30;
END_ACTION

ACTION ACT_BottleSorterVariablesWrite:
//PackMLState                         		
stBottleSorterWrite.ePackMLMode									:= P00_PackML.fbPMLModeManager.eModeStatus;
stBottleSorterWrite.ePackMLAutoState							:= P00_PackML.fbPMLAuto.ePMLState;
stBottleSorterWrite.sPackMLCommand;								 
                                 		
//stControlSignals           					
stBottleSorterWrite.bEnable										;
stBottleSorterWrite.bCycleStart									:= tpStartCycle.Q AND (NOT VIS.bCapSorterEmptyingMode OR VIS.bBottleSorterEmptyingMode) AND NOT bBottleSorterDisable;
stBottleSorterWrite.bCycleStop									:= (IbCycleStopButton AND NOT P00_PackML.tpStopCycle.Q) AND NOT VIS.bErrorOccure;													// Przepisz Stop
stBottleSorterWrite.bCycleReset									:= bCycleReseting;															// Przepisz CycleReset
stBottleSorterWrite.bManualMode									:= bManualMode;
stBottleSorterWrite.bHoming										;																		
stBottleSorterWrite.bHomingDone									;								
stBottleSorterWrite.bConfectionEnding							:= VIS.bConfectionEnding;
stBottleSorterWrite.tCycleTime									;
stBottleSorterWrite.iWatchdog									:= stBottleSorterWrite.iWatchdog + 1; 										// Do testowania komunikacji, błędu

//stError	//Przepisywane w Alarms
stBottleSorterWrite.eError.bError								:= VIS.bErrorOccure;           
stBottleSorterWrite.eError.bReset								:= bResetError;          
stBottleSorterWrite.eError.sErrorString							:= VIS.sStationErrorDescription;             
stBottleSorterWrite.eError.sStationName							:= VIS.sStationInError;     
stBottleSorterWrite.eError.nErrorCode							:= VIS.udiStationErrorCode; 

//stRecipe
stBottleSorterWrite.sRecipeName									:= sRecipeName;															//Przepisz nazwę receptury
stBottleSorterWrite.sRecipeIndex								:= sRecipeIndex;														//Przepisz index (Uwaga, String!)
                                         	                                 	
//stMachinePermissions                      	
stBottleSorterWrite.eMachinePermissions.bPermission00			;
stBottleSorterWrite.eMachinePermissions.bPermission01			;
stBottleSorterWrite.eMachinePermissions.bPermission02			;      			
stBottleSorterWrite.eMachinePermissions.bPermission03			;
stBottleSorterWrite.eMachinePermissions.bPermission04			;
stBottleSorterWrite.eMachinePermissions.bPermission05			;
stBottleSorterWrite.eMachinePermissions.bPermission06			;
stBottleSorterWrite.eMachinePermissions.bPermission07			;
//stBottleSorterWrite.eMachinePermissions.bPermission10-17

//stReservedSignals
stBottleSorterWrite.eReservedSignals.bReserved00				:= bHomingCanceled;	
stBottleSorterWrite.eReservedSignals.bReserved01				:= VIS.bBottleSorterEmptyingMode; 
stBottleSorterWrite.eReservedSignals.bReserved02				:= bHomingDialog;	
stBottleSorterWrite.eReservedSignals.bReserved03				:= IbEmergencyStop;
stBottleSorterWrite.eReservedSignals.bReserved04				:= bRecipeChangePositioning;		
stBottleSorterWrite.eReservedSignals.bReserved05				:= NOT P00_PackML.tonLongDelayAfterStart.Q OR VIS.bConfectionEnding OR VIS.bWeighingForm OR VIS.bBottleSorterHold;		
stBottleSorterWrite.eReservedSignals.bReserved06				:= IbSafetyResetIn OR QbSafetyResetBottleSorterIn OR QbSafetyResetCapSorterIn ;												
stBottleSorterWrite.eReservedSignals.bReserved07				:= VIS.bSimulation;	
stBottleSorterWrite.eReservedSignals.bReserved10				:= P00_PackML.fbbRecipeLoading.bOut; //Trwa ładowanie receptury
stBottleSorterWrite.eReservedSignals.bReserved11				:= P00_Signalization.QbStartLamp; //Miganie lampki	
stBottleSorterWrite.eReservedSignals.bReserved12				:= P00_Signalization.QbResetLamp;
stBottleSorterWrite.eReservedSignals.bReserved13				:= QbDispencersDoorsClose;			
//stBottleSorterWrite.eReservedSignals.bReserved10-17                                       					
stBottleSorterWrite.eReservedSignals.iReserved20				;                                                                                  					                      	
stBottleSorterWrite.eReservedSignals.iReserved30				;
END_ACTION

ACTION ACT_CapSorterAdsRead:
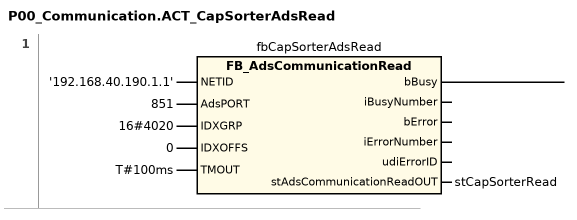
// NETWORK 1
fbCapSorterAdsRead(
    NETID := '192.168.40.190.1.1',
    AdsPORT := 851,
    IDXGRP := 16#4020,
    IDXOFFS := 0,
    TMOUT := T#100ms,
    stAdsCommunicationReadOUT => stCapSorterRead); // FB_AdsCommunicationRead
END_ACTION

ACTION ACT_CapSorterVariablesRead:
//PackMLState
stCapSorterRead.ePackMLMode;
stCapSorterRead.ePackMLAutoState;
stCapSorterRead.sPackMLCommand;                                     		
                           		
//stControlSignals        
stCapSorterRead.bEnable;      // Potrzebujemy żeby odczytać czy stacja jest włączona w recepturach 
stCapSorterRead.bCycleStart;
stCapSorterRead.bCycleStop;
stCapSorterRead.bCycleReset;
stCapSorterRead.bManualMode;
stCapSorterRead.bHoming;    // Wrote Homing przepisany w Sorterze na Read a w PackML robie bazowanie od Read
stCapSorterRead.bHomingDone;
stCapSorterRead.bConfectionEnding;
stCapSorterRead.tCycleTime;
stCapSorterRead.iWatchdog;

IF stCapSorterRead.bEnable AND NOT bCapSorterDisable THEN
	stCapSorterRead.eError.bError;
ELSE
	stCapSorterRead.eError.bError := FALSE;
END_IF

stCapSorterRead.eError.bError;
stCapSorterRead.eError.bReset;
stCapSorterRead.eError.sErrorString;
stCapSorterRead.eError.sStationName;
stCapSorterRead.eError.udiStationID;
stCapSorterRead.eError.nErrorCode;

//stRecipe
stCapSorterRead.sRecipeName;
stCapSorterRead.sRecipeIndex;
                                            	                                 	
//stMachinePermissions                      	
bCapSorterRobotPlaceDone 			:=	stCapSorterRead.eMachinePermissions.bPermission00;
bCapSorterRobotForm1CapPutted		:=	stCapSorterRead.eMachinePermissions.bPermission01;	
bCapSorterRobotForm2CapPutted		:=  stCapSorterRead.eMachinePermissions.bPermission02;	
bCapSorterRobotForm3CapPutted		:=	stCapSorterRead.eMachinePermissions.bPermission03;	
bCapSorterRobotForm4CapPutted		:=	stCapSorterRead.eMachinePermissions.bPermission04;	
bCapSorterDoor1Open					:=	NOT stCapSorterRead.eMachinePermissions.bPermission05;	
bCapSorterDoor2Open					:=	NOT stCapSorterRead.eMachinePermissions.bPermission06;	
bCapSorterDoor3Open					:=	NOT stCapSorterRead.eMachinePermissions.bPermission07;	
									//stCapSorterRead.eMachinePermissions.bPermission10-17
bCapSorterDoor4Open					:=	NOT stCapSorterRead.eMachinePermissions.bPermission10;	
bCapSorterEmergencyStopButton1Pressed:=	stCapSorterRead.eMachinePermissions.bPermission11;	
bCapSorterEmergencyStopButton2Pressed:=	stCapSorterRead.eMachinePermissions.bPermission12;	
bCapSorterEmergencyStopButton3Pressed:=	stCapSorterRead.eMachinePermissions.bPermission13;	
bCapSorterRobotPlaceAck				:=	stCapSorterRead.eMachinePermissions.bPermission14;									

//stReservedSignals
stCapSorterRead.eReservedSignals.bReserved00;// Czujnik formatki przed przeciągniem pod sorterem
stCapSorterRead.eReservedSignals.bReserved01;
stCapSorterRead.eReservedSignals.bReserved02;
stCapSorterRead.eReservedSignals.bReserved03;
stCapSorterRead.eReservedSignals.bReserved04;
stCapSorterRead.eReservedSignals.bReserved05;
QbSafetyResetCapSorterIn	:=	(stCapSorterRead.eReservedSignals.bReserved06) AND NOT bCapSorterDisable;
stCapSorterRead.eReservedSignals.bReserved07;
//stCapSorterRead.eReservedSignals.bReserved10-17
stCapSorterRead.eReservedSignals.iReserved20;//Warningi
stCapSorterRead.eReservedSignals.iReserved30;
END_ACTION

ACTION ACT_CapSorterVariablesWrite:
//PackMLState                            		
stCapSorterWrite.ePackMLMode								:= P00_PackML.fbPMLModeManager.eModeStatus;
stCapSorterWrite.ePackMLAutoState							:= P00_PackML.fbPMLAuto.ePMLState; 
stCapSorterWrite.sPackMLCommand;
              				             		
//stControlSignals  
stCapSorterWrite.bEnable									;
stCapSorterWrite.bCycleStart								:= tpStartCycle.Q AND (NOT VIS.bBottleSorterEmptyingMode OR VIS.bCapSorterEmptyingMode) AND NOT bCapSorterDisable;
stCapSorterWrite.bCycleStop									:= (IbCycleStopButton AND NOT P00_PackML.tpStopCycle.Q) AND NOT VIS.bErrorOccure;															// Przepisz Stop
stCapSorterWrite.bCycleReset								:= bCycleReseting;																// Przepisz CycleReset
stCapSorterWrite.bManualMode								:= bManualMode;
stCapSorterWrite.bHoming									;																		
stCapSorterWrite.bHomingDone								;								
stCapSorterWrite.bConfectionEnding							:= VIS.bConfectionEnding;
stCapSorterWrite.tCycleTime									;
stCapSorterWrite.iWatchdog									:= stCapSorterWrite.iWatchdog + 1; 												// Do testowania komunikacji, błędu

//stError	// Przepisywane w Alarms
stCapSorterWrite.eError.bError								:= VIS.bErrorOccure; 
stCapSorterWrite.eError.bReset								:= bResetError;    
stCapSorterWrite.eError.sErrorString						:= VIS.sStationErrorDescription;       
stCapSorterWrite.eError.sStationName						:= VIS.sStationInError;    
stCapSorterWrite.eError.nErrorCode							:= VIS.udiStationErrorCode;

//stRecipe
stCapSorterWrite.sRecipeName								:= sRecipeName;																//Przepisz nazwę receptury
stCapSorterWrite.sRecipeIndex								:= sRecipeIndex;															//Przepisz index (Uwaga, String!)
                                            	                                 	                     	
stCapSorterWrite.eMachinePermissions.bPermission00			:= bCapSorterRobotPlace; 
stCapSorterWrite.eMachinePermissions.bPermission01			:= bCapSorterRobotBottleAndNoCap1;
stCapSorterWrite.eMachinePermissions.bPermission02			:= bCapSorterRobotBottleAndNoCap2;	
stCapSorterWrite.eMachinePermissions.bPermission03			:= bCapSorterRobotBottleAndNoCap3;
stCapSorterWrite.eMachinePermissions.bPermission04			:= bCapSorterRobotBottleAndNoCap4;																						
stCapSorterWrite.eMachinePermissions.bPermission05			:= bCapSorterRobotPreparePlace;	    																		
stCapSorterWrite.eMachinePermissions.bPermission06			:= bCapSorterBeforeRobotBottleAndNoCap1;    																		
stCapSorterWrite.eMachinePermissions.bPermission07			:= bCapSorterBeforeRobotBottleAndNoCap2;  
stCapSorterWrite.eMachinePermissions.bPermission10			:= bCapSorterBeforeRobotBottleAndNoCap3;   
stCapSorterWrite.eMachinePermissions.bPermission11			:= bCapSorterBeforeRobotBottleAndNoCap4; 
																
//stCapSorterWrite.eMachinePermissions.bPermission10-17

//stReservedSignals
stCapSorterWrite.eReservedSignals.bReserved00				:= bHomingCanceled;																
stCapSorterWrite.eReservedSignals.bReserved01				:= VIS.bCapSorterEmptyingMode; 										
stCapSorterWrite.eReservedSignals.bReserved02				:= bHomingDialog;														
stCapSorterWrite.eReservedSignals.bReserved03				:= IbEmergencyStop;															
stCapSorterWrite.eReservedSignals.bReserved04				:= bRecipeChangePositioning;											
stCapSorterWrite.eReservedSignals.bReserved05				:= NOT P00_PackML.tonLongDelayAfterStart.Q;																			
stCapSorterWrite.eReservedSignals.bReserved06				:= IbSafetyResetIn OR QbSafetyResetBottleSorterIn OR QbSafetyResetCapSorterIn;																				
stCapSorterWrite.eReservedSignals.bReserved07				:= VIS.bSimulation;		
stCapSorterWrite.eReservedSignals.bReserved10				:= P00_PackML.fbbRecipeLoading.bOut; //Trwa ładowanie receptury	
stCapSorterWrite.eReservedSignals.bReserved11				:= P00_Signalization.QbStartLamp; //Miganie lampki			
stCapSorterWrite.eReservedSignals.bReserved12				:= P08_CapSorter.fbCapSorterDragStation.eRunningState >= E_DragStationState.eDraging; //Wykonywanie przeciągania, potrzebne do licznika butelek		
stCapSorterWrite.eReservedSignals.bReserved13				:= QbDispencersDoorsClose;
stCapSorterWrite.eReservedSignals.bReserved14				:= P00_Signalization.QbResetLamp;
//stCapSorterWrite.eReservedSignals.bReserved10-17
stCapSorterWrite.eReservedSignals.iReserved20				:=	VIS.iPackageHeightShow;
stCapSorterWrite.eReservedSignals.iReserved30				:= iPackageCapType;
END_ACTION

ACTION ACT_EPAdsRead:
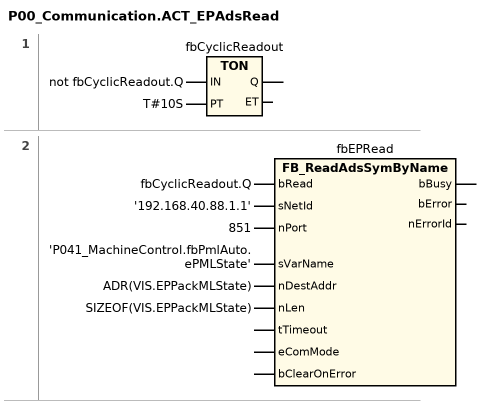
// NETWORK 1
fbCyclicReadout(IN := not fbCyclicReadout.Q, PT := T#10S); // TON

// NETWORK 2
fbEPRead(
    bRead := fbCyclicReadout.Q,
    sNetId := '192.168.40.88.1.1',
    nPort := 851,
    sVarName := 'P041_MachineControl.fbPmlAuto.ePMLState',
    nDestAddr := ADR(VIS.EPPackMLState),
    nLen := SIZEOF(VIS.EPPackMLState)); // FB_ReadAdsSymByName
END_ACTION

ACTION ACT_UPAdsRead:
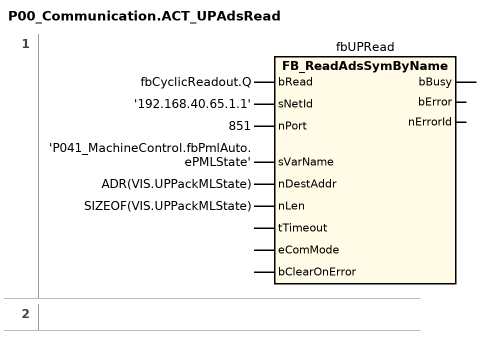
// NETWORK 1
fbUPRead(
    bRead := fbCyclicReadout.Q,
    sNetId := '192.168.40.65.1.1',
    nPort := 851,
    sVarName := 'P041_MachineControl.fbPmlAuto.ePMLState',
    nDestAddr := ADR(VIS.UPPackMLState),
    nLen := SIZEOF(VIS.UPPackMLState)); // FB_ReadAdsSymByName

// NETWORK 2
END_ACTION

END_PROGRAM

// ---- POUs/FB/ADSCommumication/FB_AdsCommunicationRead.TcPOU
FUNCTION_BLOCK FB_AdsCommunicationRead
VAR_INPUT
	NETID											: T_AmsNetID;
	AdsPORT											: T_AmsPort;
	IDXGRP											: UDINT;
	IDXOFFS											: UDINT;	
	TMOUT											: TIME;
END_VAR
VAR_OUTPUT
	bBusy											: BOOL;
	iBusyNumber 									: INT;
	bError											: BOOL;
	iErrorNumber									: INT;
	udiErrorID										: UDINT;
	stAdsCommunicationReadOUT						: ST_Communication;
END_VAR
VAR
	fbAdsCommunicationRead							: ADSREAD;			//Odczyt zmiennych 
	fbAdsReadStatus									: ADSRDSTATE;		//Odczyt stanu urządzenia ADS
	ftRead											: F_TRIG;
	bRead											: BOOL;	
	rtBusy											: R_TRIG;
	rtError											: R_TRIG;
	tonRefresh										: TON;
	udiErrorNumberTest: UDINT;
END_VAR


IF NOT bBusy AND NOT bError THEN
	bRead				:= TRUE;
END_IF
IF bError AND bRead THEN
	bRead				:= FALSE;
END_IF

ACT_AdsRead();

IF bError AND NOT bRead THEN
	bRead				:= TRUE;
END_IF

IF bRead AND NOT bError THEN
	bRead				:= FALSE;
END_IF

ACT_AdsRead();

rtBusy(CLK := bBusy);
rtError(CLK := bError);

IF rtBusy.Q THEN
    iBusyNumber                                                := iBusyNumber + 1;
    IF iBusyNumber = 32760 THEN
        iBusyNumber                                            := 0;
    END_IF
END_IF

IF rtError.Q THEN
    iErrorNumber                                                := iErrorNumber + 1;
    IF iErrorNumber = 32760 THEN
        iErrorNumber                                            := 0;
    END_IF
END_IF

IF NOT bError THEN
;	
ELSE
	;
END_IF


IF bError THEN
	udiErrorNumberTest		:= fbAdsCommunicationRead.ERRID;
END_IF

ACTION ACT_AdsRead:


fbAdsCommunicationRead(
	NETID:= 				NETID, 
	PORT:= 					AdsPORT, 
	IDXGRP:= 				IDXGRP, 
	IDXOFFS:= 				IDXOFFS, 
	LEN:= 					SIZEOF(stAdsCommunicationReadOUT), 
	DESTADDR:= 				ADR(stAdsCommunicationReadOUT), 
	READ:= 					bRead, 
	TMOUT:= 				TMOUT, 
	BUSY=> 					bBusy, 
	ERR=> 					bError, 
	ERRID=> 				udiErrorID);
END_ACTION

END_FUNCTION_BLOCK

// ---- POUs/P00_PackML.TcPOU
PROGRAM P00_PackML
VAR
	(*Pack ML v1 bloki*)
	fbPMLAuto: PS_PackML_StateMachine_Auto;
	fbPMLManual: PS_PackML_StateMachine_Manual;
	fbPMLModeManager: PS_UnitModeManager;
	
	(***PackML***)
    rtStart             		: R_TRIG; // Trigger przycisku Start cyklu
	tonStart					: TON;
    tonStarting         		: TON;	
	
    ftStopCycle         		: F_TRIG; // Trigger przycisku Stop cyklu
	rtStopCycle					: R_TRIG; // Trigger stopu cyklu
	iStoppingCase				: INT;		// Krok procedury zatrzymywania	
	tpStopCycle					: TP;
	
	rtaccelerator				: R_TRIG;
	tonFormTransporterStop		:TON;
	//koniec konfekcji
	diRFIDNumberFormatDispencerConfectionEnd	:DINT;
	bStartEndCofectionTimer		:BOOL;
	tonEndOfConfecion			:TON;
	iEndConfectionCounter		:INT;
	diPreviouslyReaded			:DINT;
	tonFormPresent				:TON;
	
    rtEstop             		: R_TRIG; // Trigger sygnalu z przekaznika bezpieczenstwa
	rtResetAlarmTrigger			: R_TRIG;
	tonResetErrorVisuCmd 		: TON;
	nResetErrorVisuCmd			: INT;
	ftVisuReset         		: F_TRIG; // Trigger komnedy Resetu z panelu wizualizacji
    rtCycleReseting     		: F_TRIG;

    tonConfectionEnding 		: TON;
	tonLongDelayAfterStart		: TON;
	ftHomingDialog				: F_TRIG;
	tofTransportersWorking		: TOF;

	bStationsAreReady			: BOOL;		// Stacje są w eReady
	bStationsAreReadyOrManual	: BOOL;		// Stacje są w eReady lub manualu
	bStationsAreManualOrError	: BOOL;
	bStationsAreReadyOrError	: BOOL;
	
	(*Filtr trybu serwisowego*)
	fbServiceMode:	FB_InputFilter;	
	
   (***** Od bazowania ****)
   	iHomingCase						   : INT;
    bHomingIsOnAtLeastOneStation       : BOOL;   //Jedna ze stacji wymaga bazowania
    bAtLeastOneOfTheStationsNeedHoming : BOOL;   //Jedna ze stacji wymaga bazowania
    rtHomingIsOnAtLeastOneStation      : R_TRIG;  //Trigger od włączenia stacji
	fbbRecipeLoading					: FB_InputFilter_v2;
	rtbRecipeLoading					: R_TRIG;
	
    (*****Pomocncze bazowanie stacji****)
	bFormsDragRightStationHommed										: BOOL;
	bFormsDragLeftStationHommed											: BOOL;
    bDispencersHommed            										: BOOL;
	bWeightLiftHommed			 										: BOOL;
	bCapPuttedCheckHommed		 										: BOOL;
	bBottleDragHommed			 										: BOOL;
    bGripperScrewerHommed        										: BOOL;
	bWickFeederHommed													: BOOL;				
	bWickFeederDragingHommed											: BOOL;		
	bLidFeederHommed													: BOOL;				
	bLidFeederDragingHommed												: BOOL;		
	bLidPuttedCheckHommed												: BOOL;			
	bLidSealerHommed													: BOOL;			
	bLidSealerDragingHommed												: BOOL;			
	bROPPFeederHommed													: BOOL;			
	bROPPDragHommed														: BOOL;			
	bROPPCappingHommed													: BOOL;			
	bCapSorterDragHommed												: BOOL;
	bCapFeederHommed													: BOOL;
	bCapCorrectCheckHommed       										: BOOL;
	bBottleTransferHommed		 										: BOOL;
	bBottleTransferAfterDragHommed 										: BOOL;
    (*****Pomocnicze stacji przesuwania****)	
	rtLongDelayFirstDraging												: R_TRIG;	
	rtLongDelayFirstDragingLidFeeder									: R_TRIG;		
	rttonLongDelayAfterStart											: R_TRIG;	
	

	
	
    (*****Pomocnicze stacji dozowania****)
    tonDelayAfterStart                : TON;
	rttonDelayAfterStart			  : R_TRIG;
	tonDispencersCase4Delay			  : TON;			
    bDelayAfterStart                  : BOOL;
    bLongDelayAfterStart              : BOOL;	
    iDispencersCase                   : INT;
    tonDosingDelay                    : TON;
    fbDispencer1BottleInCatcherSensor : FB_InputFilter;
    fbDispencer2BottleInCatcherSensor : FB_InputFilter;
    fbDispencer3BottleInCatcherSensor : FB_InputFilter;
    fbDispencer4BottleInCatcherSensor : FB_InputFilter;
    bDosingDone                       : BOOL;
	bDosingDoneFaster				  : BOOL;
    tonErrorDosing1                   : TON;
    tonErrorDosing2                   : TON;
    tonErrorDosing3                   : TON;
    tonErrorDosing4                   : TON;
    bDisp1FormsAndNoBottle            : BOOL;
    bDisp2FormsAndNoBottle            : BOOL;
    bDisp3FormsAndNoBottle            : BOOL;
    bDisp4FormsAndNoBottle            : BOOL;
    lrDosedMass1CVAux                 : LREAL; // Zmienna pomocnicza przepisywania danych dozownika 1
    lrDosedMass2CVAux                 : LREAL;
    lrDosedMass3CVAux                 : LREAL;
    lrDosedMass4CVAux                 : LREAL;
    tonCatched                        : TON;
    tonCatchNotEnable                 : TON;
    bDispencersReady                  : BOOL;
    bDispencersReadyOrSucking         : BOOL;
	bCatchersReady					  : BOOL;
	tonCatchDelay					  : TON;
	tonbDosingDone					  : TON;
	
    (*****Pomocnicze stacji wazenia****)
	fbIbWeightFirstFormSensor											: FB_InputFilter;
	fbIbWeightFirstForm2PhaseSensor										: FB_InputFilter;	
	ftfbIbWeightFirstFormSensor											: F_TRIG;
    iw1, iw2 : INT;
	tonWeightPackageState1BnCardNumber0									: TON;
	tonWeightPackageState1BnNoCardNumber								: TON;
	tonWeightPackageState2BnCardNumber0									: TON;
	tonWeightPackageState2BnNoCardNumber								: TON;
	tonWeightPackageState3BnCardNumber0									: TON;
	tonWeightPackageState3BnNoCardNumber								: TON;
	tonWeightPackageState4BnCardNumber0									: TON;
	tonWeightPackageState4BnNoCardNumber								: TON;

	tonWeightPackageState5BnCardNumber0									: TON;
	tonWeightPackageState5BnNoCardNumber								: TON;
	tonWeightPackageState6BnCardNumber0									: TON;
	tonWeightPackageState6BnNoCardNumber								: TON;
	bFormWeight1Found													: BOOL;
	bFormWeight2Found													: BOOL;
	bFormWeight3Found													: BOOL;
	bFormWeight4Found													: BOOL;
	bFormWeight5Found													: BOOL;
	bFormWeight6Found													: BOOL;
	
    (*** Pomocnicze zakręcarek  ***)	
	iGripperScrewerCase: INT;
	tonStartScrewerDelay												: TON;
	bScrewersReady														: BOOL;
	
    (*****Pomocnicze stacji sprawdzania****)
	fbIbCapPuttedCheckFormSensor										: FB_InputFilter;
	fb2IbCapPuttedCheckFormSensor										: FB_InputFilter;
	ftfbIbCapPuttedCheckFormSensor										: F_TRIG;

	rtResetAfterStart													: R_TRIG;
	rtBadBottleConvoyerStart											: R_TRIG;
	

